Yaskawa INFORM job: X2_38-47,64(2)(90,0).JBI

/JOB
//NAME X2_38-47,64(2)(90,0)
//POS
///NPOS 475,475,475,26,0,0
///TOOL 0
///POSTYPE PULSE
///PULSE
C00000=10776,-116726,-133110,-1428,79202,-268
C00001=117551,-99167,-129064,-14869,107235,-27560
C00002=118060,-97833,-124544,-14759,105287,-27149
C00003=118255,-97731,-122391,-14687,104086,-26936
C00004=118255,-99005,-121658,-14606,103015,-26804
C00005=118252,-98719,-121832,-14623,103261,-26835
C00006=118753,-92238,-119382,-14829,105109,-26899
C00007=118252,-98719,-121832,-14623,103261,-26835
C00008=117548,-101379,-128390,-14732,105732,-27372
C00009=119930,-99721,-129265,-15188,107465,-26816
C00010=120369,-98285,-124713,-15062,105542,-26424
C00011=120537,-98252,-122491,-14975,104264,-26206
C00012=120537,-99415,-121812,-14899,103281,-26083
C00013=120552,-99088,-121997,-14922,103557,-26112
C00014=120983,-92542,-119530,-15124,105413,-26206
C00015=120552,-99088,-121997,-14922,103557,-26112
C00016=119945,-101871,-128593,-15052,105999,-26622
C00017=126449,-117484,-130445,-19479,74849,-30062
C00018=126433,-122162,-123583,-20167,68593,-29001
C00019=126700,-111661,-117040,-20113,69946,-29141
C00020=126798,-108107,-114012,-20160,69935,-29102
C00021=126799,-108400,-113008,-20254,69212,-28975
C00022=126718,-108336,-113627,-20168,69582,-29070
C00023=124486,-105728,-112699,-19107,69790,-29924
C00024=126718,-108336,-113627,-20168,69582,-29070
C00025=121607,-132044,-121280,-18982,61321,-29585
C00026=106120,-105771,-112642,-10491,66484,-36125
C00027=107709,-101450,-111061,-11179,67916,-35692
C00028=106120,-105771,-112642,-10491,66484,-36125
C00029=113778,-131562,-126460,-14735,63009,-32904
C00030=125989,-135705,-128836,-15868,81833,19678
C00031=122637,-125595,-122855,-15098,82666,18409
C00032=121382,-121958,-120533,-14807,82865,17952
C00033=121382,-122071,-118910,-14836,81841,18076
C00034=121382,-121958,-120533,-14807,82865,17952
C00035=106979,-143901,-125029,-2861,68009,11090
C00036=108002,-136905,-123073,-3147,70435,11396
C00037=106979,-143901,-125029,-2861,68009,11090
C00038=130918,-93362,-108301,-23503,98063,21430
C00039=128613,-93045,-108174,-23197,97523,20724
C00040=130918,-93362,-108301,-23503,98063,21430
C00041=136165,-97259,-113946,-24281,100844,22722
C00042=136175,-89641,-119549,-25205,107565,21267
C00043=114744,-130738,-127344,18726,86415,-24127
C00044=118651,-123075,-122041,18017,86194,-22796
C00045=120132,-120263,-119410,17742,85711,-22351
C00046=120132,-120365,-118339,17753,85031,-22450
C00047=120131,-120316,-118616,17749,85218,-22423
C00048=120610,-114014,-116540,17635,86988,-22001
C00049=120131,-120316,-118616,17749,85218,-22423
C00050=120535,-116966,-117470,17658,86102,-22155
C00051=123144,-118008,-117813,17156,85246,-21372
C00052=120535,-116966,-117470,17658,86102,-22155
C00053=115268,-126863,-124750,18631,86672,-23904
C00054=115290,-123417,-132013,18678,92595,-22992
C00055=123593,-125758,-130163,-6995,115060,67946
C00056=111289,-112434,-124190,-9231,117016,63234
C00057=105837,-112853,-120878,-9823,114178,61462
C00058=105837,-113368,-119803,-9744,113264,61541
C00059=105837,-112984,-120626,-9804,113958,61481
C00060=104314,-115180,-121361,-9954,113110,60999
C00061=105837,-112984,-120626,-9804,113958,61481
C00062=140180,-156270,-135194,-3647,103600,74458
C00063=143876,-158808,-133483,-2421,103143,75779
C00064=143876,-157752,-132173,-2418,102880,75785
C00065=143876,-158999,-133717,-2421,103190,75779
C00066=142833,-166242,-135523,-2599,100548,75469
C00067=143876,-158999,-133717,-2421,103190,75779
C00068=138517,-137739,-134524,-3768,114393,73549
C00069=143641,-117492,-131018,-10110,103710,40081
C00070=127017,-112123,-129453,-9078,98380,24722
C00071=128303,-122732,-125182,-9622,82824,11347
C00072=126354,-112603,-118881,-9097,83916,10616
C00073=125631,-108986,-116438,-8904,84188,10357
C00074=125631,-109537,-114964,-8919,83013,10441
C00075=125631,-108986,-116438,-8904,84188,10357
C00076=110037,-120252,-118594,5441,76700,4050
C00077=111650,-115152,-116920,4919,78183,4659
C00078=110037,-120252,-118594,5441,76700,4050
C00079=125797,-107165,-114352,-8951,83863,10435
C00080=123589,-104463,-113383,-8361,84418,9668
C00081=125797,-107165,-114352,-8951,83863,10435
C00082=128447,-120300,-122969,-9661,82730,11402
C00083=128462,-115265,-129707,-9620,89375,10895
C00084=116938,-126430,-125851,12631,81878,-14685
C00085=119474,-116309,-119688,11957,82879,-13726
C00086=120416,-112800,-116898,11714,82830,-13413
C00087=120416,-113088,-115771,11732,82005,-13491
C00088=121130,-109897,-115487,11517,83341,-13125
C00089=121652,-107697,-114715,11371,83913,-12898
C00090=120385,-110630,-116263,11708,83544,-13356
C00091=116898,-126708,-125088,12658,81285,-14759
C00092=116961,-121523,-133241,12544,88781,-13978
C00093=110477,-156196,-127656,40514,54336,-55405
C00094=116757,-147091,-123275,37008,53079,-52657
C00095=119129,-143495,-121504,35581,52690,-51595
C00096=122199,-143523,-121511,34086,51426,-50520
C00097=119129,-143495,-121504,35581,52690,-51595
C00098=121389,-143526,-121523,34489,51757,-50806
C00099=121378,-138155,-118828,34021,52680,-50458
C00100=121389,-143526,-121523,34489,51757,-50806
C00101=121337,-120057,-120260,30579,61379,-47564
C00102=120272,-114318,-116759,30898,62447,-47698
C00103=120254,-119054,-117181,31500,60580,-48280
C00104=120272,-114318,-116759,30898,62447,-47698
C00105=110477,-159292,-131347,40206,54861,-55162
C00106=115322,-144881,-127675,10917,26238,-44128
C00107=131784,-127965,-127002,-28991,89678,-26741
C00108=120831,-123140,-121731,-27130,85392,-29797
C00109=120549,-120601,-118843,-27089,84879,-29783
C00110=120549,-120670,-117777,-27109,84260,-29640
C00111=120517,-120686,-117908,-27101,84315,-29665
C00112=120983,-114470,-115866,-27142,86197,-29928
C00113=120517,-120686,-117908,-27101,84315,-29665
C00114=121539,-130455,-126219,-27290,84728,-29379
C00115=124954,-138498,-133513,-17845,86459,-29447
C00116=125285,-130359,-127302,-17897,86875,-29392
C00117=125412,-127594,-124071,-17925,86361,-29272
C00118=125412,-127626,-123283,-17931,85883,-29202
C00119=125434,-127650,-123440,-17933,85969,-29207
C00120=125746,-120535,-121214,-17972,88215,-29428
C00121=125434,-127650,-123440,-17933,85969,-29207
C00122=125308,-130497,-125835,-17912,85951,-29248
C00123=124977,-138611,-132036,-17860,85542,-29305
C00124=131669,-108309,-130646,-31875,113573,-61343
C00125=139138,-132176,-121475,-37127,109735,-76690
C00126=136347,-141301,-121131,-36509,104575,-76083
C00127=135137,-144527,-120818,-36387,102556,-75910
C00128=135139,-143303,-118803,-36292,102059,-75739
C00129=135137,-144527,-120818,-36387,102556,-75910
C00130=123222,-117207,-112602,-33876,112841,-80142
C00131=123302,-123100,-114500,-33386,111310,-79603
C00132=123222,-117207,-112602,-33876,112841,-80142
C00133=149473,-167599,-122340,-40123,93659,-70303
C00134=145955,-169881,-122827,-40768,91382,-70949
C00135=149473,-167599,-122340,-40123,93659,-70303
C00136=154660,-158984,-124630,-39692,100555,-70658
C00137=145602,-129354,-130944,-11561,117970,-66438
C00138=141571,-135796,-129141,17923,112920,-58745
C00139=145358,-145317,-128855,18021,107261,-58200
C00140=146973,-148537,-128532,18134,105137,-57926
C00141=146977,-147425,-126561,18072,104525,-58019
C00142=146951,-147398,-126788,18082,104677,-58005
C00143=148016,-155121,-128806,18044,101844,-58047
C00144=146951,-147398,-126788,18082,104677,-58005
C00145=147811,-154474,-129578,18071,102659,-57998
C00146=150760,-151393,-128781,18698,103033,-56852
C00147=147811,-154474,-129578,18071,102659,-57998
C00148=142197,-142429,-130522,17697,110344,-58914
C00149=120703,-123129,-132845,-19094,121060,-67264
C00150=120658,-146832,-128060,-18624,118943,-66884
C00151=120634,-158899,-128202,-17585,113113,-65913
C00152=120623,-163194,-128036,-17271,110903,-65572
C00153=120623,-161024,-125795,-17237,110651,-65534
C00154=120562,-161261,-126266,-17282,110799,-65580
C00155=120543,-169070,-128088,-16945,108025,-65171
C00156=120562,-161261,-126266,-17282,110799,-65580
C00157=120603,-145779,-126506,-18564,118536,-66834
C00158=125859,-133715,-124767,-32608,106843,-81797
C00159=122845,-142953,-124347,-32149,101432,-81430
C00160=121547,-146160,-123992,-32074,99345,-81353
C00161=121546,-144979,-121994,-32008,98813,-81200
C00162=109812,-115623,-115113,-28832,111883,-86233
C00163=109420,-121759,-116943,-28463,109962,-85878
C00164=109812,-115651,-114700,-28773,111647,-86169
C00165=136113,-171916,-125823,-37236,88758,-74782
C00166=132431,-173177,-126093,-37775,86796,-75630
C00167=136113,-171916,-125823,-37236,88758,-74782
C00168=141699,-164023,-128432,-36630,95711,-74814
C00169=125872,-133752,-131219,-33440,110189,-40846
C00170=133109,-126295,-132836,-15576,121717,49477
C00171=134095,-144484,-127159,-11413,120192,39245
C00172=134095,-142728,-123587,-11251,118920,39381
C00173=134516,-141672,-122287,-11087,118973,39546
C00174=115660,-122971,-115777,13203,126220,57861
C00175=119843,-134899,-119108,17117,121012,60624
C00176=134151,-138007,-116391,34269,108686,80617
C00177=134077,-138654,-116284,35996,107959,82962
C00178=134074,-140235,-119255,36225,108790,83252
C00179=128746,-104991,-133081,28169,117444,49732
C00180=123335,-90933,-122081,14660,102496,9308
C00181=120623,-92535,-112214,7385,88125,-11837
C00182=120622,-94347,-109953,7392,85821,-11972
C00183=121302,-95773,-109518,7203,84762,-11811
C00184=119347,-92862,-108151,7759,85586,-12396
C00185=120623,-94650,-108957,7399,85059,-12018
C00186=120185,-98069,-104328,-11445,70456,7211
C00187=120621,-97250,-102226,-16251,67423,11647
C00188=120622,-96877,-104163,-16104,68755,11460
C00189=120643,-108357,-118989,-16415,66098,11840
C00190=67024,-106779,-124945,13769,92672,-20129
C00191=67015,-109280,-122780,13735,90127,-20415
C00192=69066,-117370,-123885,13251,86415,-20142
C00193=67301,-111249,-121966,13646,88610,-20491
C00194=67101,-109000,-122679,13716,90193,-20379
C00195=67110,-106486,-124839,13750,92741,-20094
C00196=120616,-103713,-129855,8435,78518,-79847
C00197=120615,-108904,-127553,8566,74477,-80127
C00198=107378,-109964,-123783,23546,74014,-82804
C00199=108339,-95722,-118664,22752,77610,-81754
C00200=115638,-127299,-133424,11228,69296,-82233
C00201=118661,-125998,-116417,35444,53464,-49551
C00202=129777,-134343,-118121,23301,43263,-42347
C00203=129442,-139718,-117663,25605,40832,-43729
C00204=126693,-153141,-115548,34897,36923,-50246
C00205=120532,-119703,-113292,30294,65799,-57942
C00206=118319,-121507,-115012,31110,66714,-58605
C00207=113281,-124998,-118777,32819,69049,-60013
C00208=113467,-117261,-128448,33027,70743,-59318
C00209=117537,-116112,-134646,12805,84442,-25722
C00210=120610,-126431,-125414,-1040,80197,-3464
C00211=120610,-126707,-122448,-1046,78230,-3447
C00212=121742,-127748,-121376,-1361,77053,-3051
C00213=120609,-128006,-121565,-1050,77021,-3438
C00214=120609,-127028,-121195,-1044,77273,-3439
C00215=120354,-127674,-120759,-4484,75447,5144
C00216=120610,-126340,-121533,-4537,76621,5189
C00217=125895,-134934,-128716,-6057,76967,6982
C00218=120648,-124280,-131590,-4464,45149,4941
C00219=120660,-101129,-132257,-5341,102721,45112
C00220=120607,-133883,-126281,-5735,119700,79532
C00221=120606,-133398,-123219,-5634,118073,79618
C00222=123085,-133870,-122397,-4740,117484,80615
C00223=120607,-133916,-122225,-5583,117200,79662
C00224=120605,-135336,-122663,-5559,116742,79683
C00225=119908,-135501,-121613,-12971,116040,68732
C00226=120606,-132780,-121444,-14001,117514,67337
C00227=120606,-133413,-124386,-14219,118956,67146
C00228=118302,-128282,-130929,-25956,92288,30440
C00229=120609,-125694,-119256,-16594,71477,14811
C00230=120609,-125321,-116628,-16727,70109,15005
C00231=120267,-125105,-115730,-16651,69613,14951
C00232=120609,-125784,-120064,8842,76919,-6014
C00233=120609,-126092,-120067,8848,76762,-6022
C00234=120946,-125981,-118164,18196,76467,-19006
C00235=120609,-125456,-118894,18238,77226,-19012
C00236=120610,-125544,-121647,18141,78796,-18775
C00237=120644,-111765,-129409,18832,94472,-5338
C00238=120647,-108820,-131188,26213,120818,60808
C00239=120603,-141811,-125437,24145,112419,84195
C00240=120603,-140407,-122244,23914,111279,83943
C00241=120885,-139622,-121239,23950,111003,83997
C00242=120603,-141924,-124431,0,115210,75490
C00243=120602,-141703,-124653,2,115461,75491
C00244=121293,-137419,-119128,-26325,110161,66441
C00245=120602,-139074,-119094,-30337,107734,65073
C00246=120603,-140473,-121905,-30531,108612,64825
C00247=123038,-137969,-128708,-31970,112888,64779
C00248=147472,-118060,-121113,-40576,103304,81843
C00249=147472,-118630,-118217,-40218,101703,82475
C00250=147472,-118727,-117017,-40094,101093,82713
C00251=147408,-115266,-125424,-616,120610,87255
C00252=147440,-115512,-125518,-608,120541,87267
C00253=147454,-115617,-125558,-7144,119076,75809
C00254=147463,-115686,-125590,-12209,115534,64774
C00255=147467,-115708,-125608,-15036,110623,54333
C00256=147465,-115687,-125611,-15580,106535,46817
C00257=147461,-115654,-125607,-15271,104034,42312
C00258=147458,-115622,-125603,-14500,101619,37854
C00259=147455,-115603,-125598,-14501,101625,37852
C00260=147455,-114670,-126645,-14574,102714,37720
C00261=147454,-112308,-128585,-14752,105047,37432
C00262=120607,-127649,-132770,5702,79300,-5510
C00263=120610,-123519,-126906,5727,77820,-5577
C00264=120610,-124347,-124400,5769,75861,-5668
C00265=121896,-125923,-123599,5365,74477,-5288
C00266=120260,-126985,-123973,12405,76553,-12588
C00267=120608,-127390,-125694,8862,79219,-9976
C00268=120607,-127434,-125218,-886,76106,-6932
C00269=120607,-127109,-124972,1540,76154,-9484
C00270=116410,-121243,-123100,2858,78131,-10867
C00271=112513,-116509,-121595,4066,79794,-12120
C00272=109281,-113129,-120468,5058,81013,-13145
C00273=120610,-123835,-125318,1528,78049,-9462
C00274=120610,-122990,-127374,1521,79748,-9441
C00275=-2000,-133752,-131219,0,47993,0
C00276=63459,-114373,-79771,-19626,40886,-37257
C00277=120535,72123,63468,-4767,55280,-66520
C00278=120830,77643,74299,-5152,51483,-66214
C00279=120946,80397,79380,-5338,49786,-66073
C00280=120946,82340,83558,-5464,48220,-65985
C00281=120946,80397,79380,-5338,49786,-66073
C00282=120262,74330,73734,-4961,50098,-66387
C00283=120723,78845,79280,-5280,49039,-66130
C00284=120262,74330,73734,-4961,50098,-66387
C00285=120141,71846,69055,-4791,51689,-66517
C00286=119837,66739,58851,-4430,55315,-66806
C00287=133022,42927,30487,-538,57153,-74648
C00288=133254,46148,37978,-681,54200,-74537
C00289=133346,47607,41185,-741,52977,-74490
C00290=133347,48340,43676,-753,51820,-74481
C00291=133346,47607,41185,-741,52977,-74490
C00292=132762,43480,38515,-427,52495,-74733
C00293=133123,46716,41988,-628,52023,-74578
C00294=132762,43480,38515,-427,52495,-74733
C00295=132666,42024,35338,-369,53702,-74778
C00296=132425,38795,27897,-232,56620,-74884
C00297=155117,742,-2384,-2320,66217,-73300
C00298=180906,93001,78797,-1706,80780,-74950
C00299=182918,91178,77459,-1890,80713,-74262
C00300=182918,92061,79857,-1895,79691,-74247
C00301=182918,93168,82666,-1899,78530,-74228
C00302=182918,93037,82343,-1899,78661,-74230
C00303=183042,90194,78719,-1906,79434,-74200
C00304=182918,91730,78973,-1891,80062,-74252
C00305=174748,66441,50706,-1110,84503,-77209
C00306=160848,12597,380,297,58397,-81989
C00307=166181,24822,19162,1318,68440,4797
C00308=165629,32403,32901,1529,63893,4538
C00309=165325,34741,37059,1643,62541,4405
C00310=165325,35383,38873,1654,61756,4395
C00311=165325,34741,37059,1643,62541,4405
C00312=165316,38003,40423,1653,62149,4395
C00313=165325,34741,37059,1643,62541,4405
C00314=158615,42058,44677,13811,65940,-11748
C00315=158695,42833,46513,13869,65215,-11806
C00316=159268,43921,47675,13753,64967,-11620
C00317=158695,42064,44447,13779,66066,-11705
C00318=158695,37647,30177,13233,72407,-10974
C00319=159201,26732,24188,1278,51025,-82719
C00320=159224,30548,32077,1320,48132,-82748
C00321=159868,34226,37454,953,46702,-82474
C00322=159868,34770,38966,962,46052,-82480
C00323=159702,29671,32865,1045,47189,-82543
C00324=159324,28280,32585,1288,46650,-82722
C00325=159393,32989,37300,1258,46169,-82698
C00326=159613,30008,32996,1100,47283,-82582
C00327=159229,22535,21884,1275,50287,-82716
C00328=183717,62399,62329,-13487,47753,-71656
C00329=183547,68974,74327,-14313,43831,-71133
C00330=183480,72253,80019,-14758,42056,-70865
C00331=183483,74717,84855,-15260,40402,-70564
C00332=183480,72253,80019,-14758,42056,-70865
C00333=183942,65201,73380,-14911,42587,-70727
C00334=183665,70044,79187,-15050,41486,-70670
C00335=183942,65201,73380,-14911,42587,-70727
C00336=184013,62287,68228,-14508,44220,-70970
C00337=184190,56247,57052,-13734,47916,-71463
C00338=194866,74493,66336,-18454,53556,-67625
C00339=193573,89765,89535,-19520,47162,-66942
C00340=193573,91648,93222,-19932,45935,-66672
C00341=193573,93286,96299,-20287,44943,-66446
C00342=193573,92255,94376,-20065,45559,-66588
C00343=194136,78940,77511,-19269,49033,-67072
C00344=194228,80437,80064,-19546,48302,-66875
C00345=193714,88383,90097,-19926,46207,-66663
C00346=194171,78002,75688,-19109,49654,-67182
C00347=183631,19122,4613,-11412,60722,-73268
C00348=122649,-90706,-82561,19496,61180,-53724
C00349=122649,-90706,-82561,19496,61180,-53724
C00350=146927,-106152,-71782,9593,42642,-76873
C00351=147684,-69879,-51768,13743,41767,-65179
C00352=150199,4793,-22546,4300,98283,-83429
C00353=150319,1938,-15262,4232,92343,-83591
C00354=150367,1184,-14302,4224,91365,-83608
C00355=150367,1240,-12851,4221,90502,-83638
C00356=150367,1184,-14302,4224,91365,-83608
C00357=150123,10711,-6542,4244,91496,-83686
C00358=150277,8779,-6240,4228,90310,-83676
C00359=150175,6887,-7898,4237,90361,-83709
C00360=149968,8102,-7784,4257,90924,-83760
C00361=150441,9583,-10879,4230,93564,-83509
C00362=131878,-32966,-47472,26236,62495,-86167
C00363=135680,-27941,-40403,24709,59747,-85262
C00364=135680,-27934,-39056,24908,58995,-85442
C00365=135680,-27896,-37768,25103,58290,-85615
C00366=135677,-27936,-39177,24874,59064,-85427
C00367=134264,-34276,-43444,25765,58916,-86062
C00368=134265,-34195,-41853,26012,58067,-86277
C00369=135346,-30088,-39110,25338,58118,-85800
C00370=135733,-34145,-44672,24799,59221,-85365
C00371=145616,-30275,-43889,19038,58025,-81528
C00372=147684,-69879,-51768,13743,41767,-65179
C00373=146927,-106152,-71782,9593,42642,-76873
C00374=150216,-104680,-71296,7403,42753,-75254
C00375=181592,-40940,-51538,-10072,64088,-74364
C00376=161871,19225,13725,-11181,66080,-79002
C00377=161452,20882,19453,-11278,63397,-78896
C00378=164352,10606,16407,-20315,52242,-75889
C00379=162815,10479,16392,-19594,51818,-76493
C00380=160145,20957,19678,-10844,63120,-79369
C00381=160561,19267,13917,-10753,65806,-79466
C00382=160561,19267,13917,-10683,67653,-23343
C00383=154925,6937,8528,5000,60577,-30889
C00384=159657,9316,12490,-1477,58995,-24503
C00385=156738,10623,15910,1856,57584,-27775
C00386=156328,10923,16900,2033,57138,-27949
C00387=155501,5675,10762,2341,58239,-28253
C00388=164062,6293,11536,-10601,60711,-458
C00389=163435,22729,32465,-8745,61137,-855
C00390=168216,43762,52548,-18935,71405,19387
C00391=169763,36380,39766,-18709,75622,19280
C00392=165018,20718,26071,-18440,72235,15535
C00393=160304,21163,32931,-8111,30161,-79764
C00394=160077,26796,41073,-8391,28042,-79637
C00395=159587,29219,48591,-14117,21277,-77933
C00396=162103,29346,48721,-18047,21745,-75808
C00397=162103,29346,48721,-18047,21745,-75808
C00398=160812,19418,34049,-13727,25286,-78018
C00399=165374,24294,37670,-31515,32350,-71401
C00400=161014,23173,34950,10300,28145,-85028
C00401=161267,29296,43834,10809,25831,-85265
C00402=163117,31582,50788,6969,18892,-84323
C00403=165058,31936,51150,3284,18732,-82405
C00404=165058,31936,51150,3284,18732,-82405
C00405=165058,26028,37877,2608,23858,-82083
C00406=156219,-6549,3189,13376,29320,-87906
C00407=193662,52178,54811,-23966,35939,-65070
C00408=193395,59348,65976,-25679,32954,-64157
C00409=193846,66406,75330,-27317,31216,-63316
C00410=195732,71420,81412,-29926,30818,-61781
C00411=190088,34040,27543,-17579,42098,-68896
C00412=195743,56061,59163,-26082,35942,-63785
C00413=183848,81700,74678,1498,72719,-73637
C00414=175309,68305,57984,16674,76256,-76182
C00415=174796,71984,66825,17009,72957,-76836
C00416=176911,74218,69518,16737,72030,-76191
C00417=175436,69064,60684,16741,75010,-76311
C00418=157840,39389,32444,18807,80897,-81798
C00419=152544,-11566,-20773,-4534,70818,-69047
C00420=121453,69600,74634,-8596,44521,-67329
C00421=121610,79178,90779,-9562,39584,-66727
C00422=122256,62901,78801,-13281,29449,-64716
C00423=119976,69596,87112,-11678,27131,-65794
C00424=119487,82929,95001,-8292,38695,-67720
C00425=113080,77640,80749,10055,45502,-72493
C00426=113679,80944,85852,9958,44007,-72378
C00427=115090,79143,84432,3405,41517,-71194
C00428=114991,50178,46533,3890,43654,-71191
C00429=130022,56817,59683,7064,48325,-77006
C00430=130464,62791,70833,7260,44523,-77097
C00431=132030,55766,67561,6192,36406,-76838
C00432=136266,49513,60493,2695,37313,-74483
C00433=134997,54946,61777,4491,45732,-74911
C00434=138242,-4678,-14452,2133,61853,-73053
C00435=140332,-41635,-35386,1385,55778,-72457
C00436=125234,-105855,-90971,8573,57832,-78294
C00437=134723,-30987,-43000,16193,82094,73445
C00438=147286,-18641,-32771,-2207,85620,76456
C00439=145565,-8574,-24761,171,91849,76015
C00440=144872,-8220,-24480,237,91860,75784
C00441=148310,-19029,-33055,-2389,85623,76796
C00442=149415,-19533,-33424,-2584,85625,77164
C00443=149671,-4054,-21067,1311,92603,77409
C00444=148276,-3677,-20761,1434,92631,76943
C00445=148276,-3408,-24949,1441,95347,76974
C00446=162074,-26616,-42506,1763,64705,79693
C00447=162070,-24854,-37261,1799,62384,79656
C00448=162588,-20391,-33053,1539,62074,79844
C00449=161725,-20523,-33128,1979,62071,79525
C00450=159769,-24818,-37192,4027,62449,78761
C00451=159682,-26579,-42435,3993,64769,78811
C00452=159749,-26590,-42466,830,64636,81339
C00453=159773,-24828,-37221,834,62313,81331
C00454=157385,-24447,-34130,6743,58116,80693
C00455=158588,-24538,-34197,6069,58011,81159
C00456=162116,-24842,-37231,-1419,62318,82243
C00457=162183,-26603,-42475,-1425,64641,82238
C00458=125234,-105855,-90971,8573,57832,-78294
C00459=122641,-148463,-123471,10002,56262,-79479
C00460=122641,-148463,-123471,10002,56262,-79479
C00461=171100,-2344,-14517,-1298,46918,-78414
C00462=177009,29876,35461,-7963,33075,-74566
C00463=175070,31868,42315,2631,27249,-76698
C00464=178558,34317,44810,-1908,26956,-74189
C00465=176419,28474,30454,-160,33043,-75584
C00466=173102,47124,36593,11518,57062,-77684
C00467=172903,62994,47851,2783,78849,-77249
C00468=172923,63788,52294,3178,77603,-77352
C00469=170832,85464,80401,8251,77478,-78178
C00470=174864,89706,85780,7992,75954,-76876
C00471=176408,69063,51861,3929,81897,-76013
C00472=176687,67050,51974,2579,79340,-76016
C00473=124677,13030,-21056,9614,100342,-34470
C00474=10907,-117335,-90652,18762,63715,59495
BC00000=165804,522273,1075193
BC00001=398158,179848,1075139
BC00002=398158,179848,1075139
BC00003=398158,179848,1075139
BC00004=398158,179848,1075139
BC00005=398158,179848,1075139
BC00006=398158,179848,1075139
BC00007=398158,179848,1075139
BC00008=398158,179848,1075139
BC00009=355141,187784,1075139
BC00010=355141,187784,1075139
BC00011=355141,187784,1075139
BC00012=355141,187784,1075139
BC00013=355141,187784,1075139
BC00014=355141,187784,1075139
BC00015=355141,187784,1075139
BC00016=355141,187784,1075139
BC00017=253971,280733,1075139
BC00018=253971,280733,1075139
BC00019=253971,280733,1075139
BC00020=253971,280733,1075139
BC00021=253971,280733,1075139
BC00022=253971,280733,1075139
BC00023=253971,280733,1075139
BC00024=253971,280733,1075139
BC00025=253971,280733,1075139
BC00026=253971,280733,1075139
BC00027=253971,280733,1075139
BC00028=253971,280733,1075139
BC00029=253971,280733,1075139
BC00030=147021,241254,1075139
BC00031=147021,241254,1075139
BC00032=147021,241254,1075139
BC00033=147021,241254,1075139
BC00034=147021,241254,1075139
BC00035=147021,241254,1075139
BC00036=147021,241254,1075139
BC00037=147021,241254,1075139
BC00038=147021,241254,1075139
BC00039=147021,241254,1075139
BC00040=147021,241254,1075139
BC00041=147021,241254,1075139
BC00042=147021,241254,1075139
BC00043=175602,243488,1075139
BC00044=175602,243488,1075139
BC00045=175602,243488,1075139
BC00046=175602,243488,1075139
BC00047=175602,243488,1075139
BC00048=175602,243488,1075139
BC00049=175602,243488,1075139
BC00050=175602,243488,1075139
BC00051=175602,243488,1075139
BC00052=175602,243488,1075139
BC00053=175602,243488,1075139
BC00054=175602,243488,1075139
BC00055=144296,215160,1075139
BC00056=144296,215160,1075139
BC00057=144296,215160,1075139
BC00058=144296,215160,1075139
BC00059=144296,215160,1075139
BC00060=144296,215160,1075139
BC00061=144296,215160,1075139
BC00062=144296,215160,1075139
BC00063=144296,215160,1075139
BC00064=144296,215160,1075139
BC00065=144296,215160,1075139
BC00066=144296,215160,1075139
BC00067=144296,215160,1075139
BC00068=144296,215160,1075139
BC00069=159912,261457,1075139
BC00070=164424,314586,1075139
BC00071=171018,327464,1075139
BC00072=171018,327464,1075139
BC00073=171018,327464,1075139
BC00074=171018,327464,1075139
BC00075=171018,327464,1075139
BC00076=171018,327464,1075139
BC00077=171018,327464,1075139
BC00078=171018,327464,1075139
BC00079=171018,327464,1075139
BC00080=171018,327464,1075139
BC00081=171018,327464,1075139
BC00082=171018,327464,1075139
BC00083=171018,327464,1075139
BC00084=164722,348126,1075139
BC00085=164722,348126,1075139
BC00086=164722,348126,1075139
BC00087=164722,348126,1075139
BC00088=164722,348126,1075139
BC00089=164722,348126,1075139
BC00090=164722,348126,1075139
BC00091=164722,348126,1075139
BC00092=164722,348126,1075139
BC00093=143323,255421,1075139
BC00094=143323,255421,1075139
BC00095=143323,255421,1075139
BC00096=143323,255421,1075139
BC00097=143323,255421,1075139
BC00098=143323,255421,1075139
BC00099=143323,255421,1075139
BC00100=143323,255421,1075139
BC00101=143323,255421,1075139
BC00102=143323,255421,1075139
BC00103=143323,255421,1075139
BC00104=143323,255421,1075139
BC00105=143323,255421,1075139
BC00106=95176,326084,1075139
BC00107=33051,239015,1075139
BC00108=33051,239015,1075139
BC00109=33051,239015,1075139
BC00110=33051,239015,1075139
BC00111=33051,239015,1075139
BC00112=33051,239015,1075139
BC00113=33051,239015,1075139
BC00114=33051,239015,1075139
BC00115=1592,244787,1075139
BC00116=1592,244787,1075139
BC00117=1592,244787,1075139
BC00118=1592,244787,1075139
BC00119=1592,244787,1075139
BC00120=1592,244787,1075139
BC00121=1592,244787,1075139
BC00122=1592,244787,1075139
BC00123=1592,244787,1075139
BC00124=16444,332290,1075139
BC00125=28284,383081,1075139
BC00126=28284,383081,1075139
BC00127=28284,383081,1075139
BC00128=28284,383081,1075139
BC00129=28284,383081,1075139
BC00130=28284,383081,1075139
BC00131=28284,383081,1075139
BC00132=28284,383081,1075139
BC00133=28284,383081,1075139
BC00134=28284,383081,1075139
BC00135=28284,383081,1075139
BC00136=28284,383081,1075139
BC00137=49933,363253,1075139
BC00138=70307,361243,1075139
BC00139=70307,361243,1075139
BC00140=70307,361243,1075139
BC00141=70307,361243,1075139
BC00142=70307,361243,1075139
BC00143=70307,361243,1075139
BC00144=70307,361243,1075139
BC00145=70307,361243,1075139
BC00146=70307,361243,1075139
BC00147=70307,361243,1075139
BC00148=70307,361243,1075139
BC00149=113384,373634,1075139
BC00150=113384,343814,1075139
BC00151=113384,343814,1075139
BC00152=113384,343814,1075139
BC00153=113384,343814,1075139
BC00154=113384,343814,1075139
BC00155=113384,343814,1075139
BC00156=113384,343814,1075139
BC00157=113384,343814,1075139
BC00158=126163,380629,1075139
BC00159=126163,380629,1075139
BC00160=126163,380629,1075139
BC00161=126163,380629,1075139
BC00162=126163,380629,1075139
BC00163=126163,380629,1075139
BC00164=126163,380629,1075139
BC00165=126163,380629,1075139
BC00166=126163,380629,1075139
BC00167=126163,380629,1075139
BC00168=126163,380629,1075139
BC00169=126163,380629,1075139
BC00170=153244,197421,1075139
BC00171=154878,181155,1075139
BC00172=159551,183681,1075139
BC00173=161025,184477,1075133
BC00174=188164,185165,1075136
BC00175=159382,201380,1075135
BC00176=196155,204160,1075132
BC00177=201120,202214,1075139
BC00178=203654,196593,1075139
BC00179=184090,265203,1075139
BC00180=164129,334283,1075139
BC00181=154120,368924,1075139
BC00182=151898,363919,1075139
BC00183=151009,361917,1075139
BC00184=151009,361917,1075139
BC00185=197558,335778,1075139
BC00186=159988,349936,1075139
BC00187=151141,355258,1075139
BC00188=148277,361304,1075139
BC00189=148277,361304,1075139
BC00190=312259,195594,1075139
BC00191=311963,190251,1075139
BC00192=311844,188113,1075139
BC00193=362717,179281,1075128
BC00194=362836,181418,1075139
BC00195=363132,186762,1075139
BC00196=102779,255305,1075139
BC00197=101436,253332,1075139
BC00198=100899,252542,1075139
BC00199=100899,252542,1075139
BC00200=101410,246391,1075139
BC00201=141499,261853,1075139
BC00202=141499,261853,1075139
BC00203=141499,261853,1075139
BC00204=141499,261852,1075136
BC00205=141499,261853,1075139
BC00206=141499,261853,1075139
BC00207=141499,261853,1075139
BC00208=141499,274005,1075139
BC00209=68111,269753,1075139
BC00210=16814,266781,1075139
BC00211=16546,261584,1075139
BC00212=16439,259506,1075139
BC00213=16439,259506,1075139
BC00214=71877,249918,1075139
BC00215=67448,250953,1075139
BC00216=67006,253063,1075139
BC00217=65899,258340,1075139
BC00218=65899,288131,1075139
BC00219=98307,337973,1075139
BC00220=125063,358885,1075139
BC00221=125778,364300,1075139
BC00222=126063,366466,1075139
BC00223=130842,366450,1075139
BC00224=170092,366314,1075137
BC00225=159428,366441,1075139
BC00226=156853,364418,1075139
BC00227=154110,359318,1075139
BC00228=114676,288419,1075139
BC00229=142986,258877,1075139
BC00230=146299,253666,1075139
BC00231=147625,251582,1075139
BC00232=194925,245639,1075139
BC00233=156825,252253,1075139
BC00234=172687,249256,1075139
BC00235=174276,250992,1075139
BC00236=178251,255331,1075139
BC00237=164902,278776,1075139
BC00238=91091,340629,1075139
BC00239=59682,360606,1075139
BC00240=57241,365786,1075139
BC00241=56264,367859,1075139
BC00242=29820,362432,1075139
BC00243=76738,362270,1075139
BC00244=34590,371298,1075139
BC00245=25837,371005,1075139
BC00246=21253,366566,1075139
BC00247=34673,355700,1075135
BC00248=267722,172731,1075139
BC00249=272714,174556,1075139
BC00250=274711,175286,1075139
BC00251=328692,136963,1075139
BC00252=294146,156358,1075139
BC00253=279419,165219,1075139
BC00254=269323,178854,1075139
BC00255=265414,195151,1075139
BC00256=267320,208388,1075139
BC00257=271316,217638,1075139
BC00258=275010,224166,1075139
BC00259=277506,226556,1075139
BC00260=275846,227409,1075139
BC00261=272525,229113,1075139
BC00262=271699,297736,1073424
BC00263=294810,273775,1075139
BC00264=293529,268177,1075139
BC00265=293016,265937,1075139
BC00266=307027,261102,1075139
BC00267=302570,257740,1075139
BC00268=285679,262491,1075139
BC00269=319740,246081,1075139
BC00270=320984,245484,1075139
BC00271=320984,245484,1075139
BC00272=320984,245484,1075139
BC00273=325754,245581,1075139
BC00274=326738,249882,1075139
BC00275=126163,523905,1075139
BC00276=216710,557083,641270
BC00277=301352,400556,286994
BC00278=301352,400556,286994
BC00279=301352,400556,286994
BC00280=301352,400556,286994
BC00281=301352,400556,286994
BC00282=301352,400556,286994
BC00283=301352,400556,286994
BC00284=301352,400556,286994
BC00285=301352,400556,286994
BC00286=301352,400556,286994
BC00287=314469,400556,277493
BC00288=314469,400556,277493
BC00289=314469,400556,277493
BC00290=314469,400556,277493
BC00291=314469,400556,277493
BC00292=314469,400556,277493
BC00293=314469,400556,277493
BC00294=314469,400556,277493
BC00295=314469,400556,277493
BC00296=314469,400556,277493
BC00297=331599,400556,395859
BC00298=359853,392268,238433
BC00299=359853,392268,238433
BC00300=359853,392268,238433
BC00301=359853,392268,238433
BC00302=359853,392268,238433
BC00303=359853,392268,238433
BC00304=359853,392268,238433
BC00305=343262,398138,316204
BC00306=345835,406354,335171
BC00307=345835,406354,335171
BC00308=345835,406354,335171
BC00309=344242,406354,335171
BC00310=344242,406354,335171
BC00311=344242,406354,335171
BC00312=344242,406354,335171
BC00313=344242,406354,335171
BC00314=344242,406354,335171
BC00315=344242,406354,335171
BC00316=344242,406354,335171
BC00317=344242,406354,335171
BC00318=344242,406354,335171
BC00319=319771,400556,337896
BC00320=319771,400556,337896
BC00321=319771,400556,337896
BC00322=319771,400556,337896
BC00323=319771,400556,337896
BC00324=319771,400556,337896
BC00325=319771,400556,337896
BC00326=319771,400556,337896
BC00327=319771,400556,337896
BC00328=359948,400556,338029
BC00329=359948,400556,338029
BC00330=358355,400556,338029
BC00331=358355,400556,338029
BC00332=358355,400556,338029
BC00333=358355,400556,338029
BC00334=358355,400556,338029
BC00335=358355,400556,338029
BC00336=358355,400556,338029
BC00337=358355,400556,338029
BC00338=365219,400556,270898
BC00339=365219,400556,270898
BC00340=365219,400556,270898
BC00341=365219,400556,270898
BC00342=365219,400556,270898
BC00343=365219,400556,270898
BC00344=365218,400556,270894
BC00345=365218,400556,270894
BC00346=365218,400556,270894
BC00347=365219,411738,375837
BC00348=329511,449778,412801
BC00349=329511,557326,412801
BC00350=219184,520233,311741
BC00351=202274,450326,276450
BC00352=161102,424985,263657
BC00353=161102,424985,263657
BC00354=161102,424985,263657
BC00355=161102,424985,263657
BC00356=161102,424985,263657
BC00357=161102,424985,263657
BC00358=161102,424985,263657
BC00359=161102,424985,263657
BC00360=161102,424985,263657
BC00361=161102,424985,263657
BC00362=144242,432455,148407
BC00363=144242,432455,148407
BC00364=144242,432455,148407
BC00365=144242,432455,148407
BC00366=144243,432453,148404
BC00367=144243,432453,148404
BC00368=144243,432453,148404
BC00369=144243,432453,148404
BC00370=144243,432453,148404
BC00371=179284,432455,148407
BC00372=202274,450326,276450
BC00373=219184,520233,311741
BC00374=365219,520233,600293
BC00375=365219,400556,421118
BC00376=312291,400556,335654
BC00377=312291,400556,335654
BC00378=312291,400556,335654
BC00379=312291,400556,335654
BC00380=312291,400556,335654
BC00381=312291,400556,335654
BC00382=312291,400556,335654
BC00383=312291,400556,335654
BC00384=312291,400556,335654
BC00385=312291,400556,335654
BC00386=312291,400556,335654
BC00387=312291,400556,335654
BC00388=312291,400556,335654
BC00389=312291,400556,375436
BC00390=311759,400169,372248
BC00391=311759,400169,372248
BC00392=312261,400534,445273
BC00393=315262,415157,353191
BC00394=315262,415157,353191
BC00395=315262,415157,353191
BC00396=315262,415157,353191
BC00397=315262,415157,353191
BC00398=315262,415157,353191
BC00399=315262,415157,353191
BC00400=349728,401236,343133
BC00401=349728,401236,343133
BC00402=349728,401236,343133
BC00403=349728,401236,343133
BC00404=349728,401236,343133
BC00405=349728,401236,343133
BC00406=329311,401236,343133
BC00407=366682,400556,290774
BC00408=366682,400556,290774
BC00409=366681,400557,290771
BC00410=366681,400557,290771
BC00411=353522,400557,312772
BC00412=366682,400556,290774
BC00413=341680,400556,335831
BC00414=329114,400556,286060
BC00415=329114,400556,286060
BC00416=329114,400556,286060
BC00417=329114,400556,286060
BC00418=329114,400556,391747
BC00419=306068,400556,345190
BC00420=296056,400556,352007
BC00421=296056,400556,352007
BC00422=296056,400556,352007
BC00423=296056,400556,352007
BC00424=296056,400556,352007
BC00425=296056,400556,305429
BC00426=296056,400556,299166
BC00427=296056,400556,299166
BC00428=296056,400556,299166
BC00429=322956,400556,356242
BC00430=322956,400556,356242
BC00431=322956,400556,356242
BC00432=322956,400556,356242
BC00433=322956,400556,356242
BC00434=323481,404427,418512
BC00435=346006,570548,634248
BC00436=182874,521648,141172
BC00437=138881,416921,238060
BC00438=138881,416921,238060
BC00439=138881,416921,238060
BC00440=138881,416921,238060
BC00441=138881,416921,238060
BC00442=138881,416921,238060
BC00443=147186,418329,239646
BC00444=147186,418329,239646
BC00445=147186,418329,239646
BC00446=187699,415530,182613
BC00447=187699,415530,182613
BC00448=187699,415530,182613
BC00449=187699,415530,182613
BC00450=187699,415530,182613
BC00451=187699,415530,182613
BC00452=187889,415612,182576
BC00453=187889,415612,182576
BC00454=187889,415612,182576
BC00455=187889,415612,182576
BC00456=187889,415612,182576
BC00457=187889,415612,182576
BC00458=182874,521648,141172
BC00459=322956,521648,357949
BC00460=322956,420180,357949
BC00461=348415,400556,248672
BC00462=348415,400556,302439
BC00463=348415,400556,302439
BC00464=348415,400556,302439
BC00465=348415,400556,302439
BC00466=348415,400556,302439
BC00467=339822,400556,351764
BC00468=339562,400556,281997
BC00469=339562,400556,281997
BC00470=339562,400556,281997
BC00471=339562,400556,281997
BC00472=339562,400556,330065
BC00473=340056,504795,481042
BC00474=165804,522273,534000
EC00000=-798156,-183832
EC00001=-798156,-183832
EC00002=-798156,-183832
EC00003=-798156,-183832
EC00004=-798156,-183832
EC00005=-798156,-183832
EC00006=-798156,-183832
EC00007=-798156,-183832
EC00008=-798156,-183832
EC00009=-798156,-183832
EC00010=-798156,-183832
EC00011=-798156,-183832
EC00012=-798156,-183832
EC00013=-798156,-183832
EC00014=-798156,-183832
EC00015=-798156,-183832
EC00016=-798156,-183832
EC00017=-798156,-183832
EC00018=-798156,-183832
EC00019=-798156,-183832
EC00020=-798156,-183832
EC00021=-798156,-183832
EC00022=-798156,-183832
EC00023=-798156,-183832
EC00024=-798156,-183832
EC00025=-798156,-183832
EC00026=-798156,-183832
EC00027=-798156,-183832
EC00028=-798156,-183832
EC00029=-798156,-183832
EC00030=-798156,-183832
EC00031=-798156,-183832
EC00032=-798156,-183832
EC00033=-798156,-183832
EC00034=-798156,-183832
EC00035=-798156,-183832
EC00036=-798156,-183832
EC00037=-798156,-183832
EC00038=-798156,-183832
EC00039=-798156,-183832
EC00040=-798156,-183832
EC00041=-798156,-183832
EC00042=-798156,-183832
EC00043=-798156,-183832
EC00044=-798156,-183832
EC00045=-798156,-183832
EC00046=-798156,-183832
EC00047=-798156,-183832
EC00048=-798156,-183832
EC00049=-798156,-183832
EC00050=-798156,-183832
EC00051=-798156,-183832
EC00052=-798156,-183832
EC00053=-798156,-183832
EC00054=-798156,-183832
EC00055=-798156,-183832
EC00056=-798156,-183832
EC00057=-798156,-183832
EC00058=-798156,-183832
EC00059=-798156,-183832
EC00060=-798156,-183832
EC00061=-798156,-183832
EC00062=-798156,-183832
EC00063=-798156,-183832
EC00064=-798156,-183832
EC00065=-798156,-183832
EC00066=-798156,-183832
EC00067=-798156,-183832
EC00068=-798156,-183832
EC00069=-798156,-183832
EC00070=-798156,-183832
EC00071=-798156,-183832
EC00072=-798156,-183832
EC00073=-798156,-183832
EC00074=-798156,-183832
EC00075=-798156,-183832
EC00076=-798156,-183832
EC00077=-798156,-183832
EC00078=-798156,-183832
EC00079=-798156,-183832
EC00080=-798156,-183832
EC00081=-798156,-183832
EC00082=-798156,-183832
EC00083=-798156,-183832
EC00084=-798156,-183832
EC00085=-798156,-183832
EC00086=-798156,-183832
EC00087=-798156,-183832
EC00088=-798156,-183832
EC00089=-798156,-183832
EC00090=-798156,-183832
EC00091=-798156,-183832
EC00092=-798156,-183832
EC00093=-798156,-183832
EC00094=-798156,-183832
EC00095=-798156,-183832
EC00096=-798156,-183832
EC00097=-798156,-183832
EC00098=-798156,-183832
EC00099=-798156,-183832
EC00100=-798156,-183832
EC00101=-798156,-183832
EC00102=-798156,-183832
EC00103=-798156,-183832
EC00104=-798156,-183832
EC00105=-798156,-183832
EC00106=-798156,-183832
EC00107=-798156,-183832
EC00108=-798156,-183832
EC00109=-798156,-183832
EC00110=-798156,-183832
EC00111=-798156,-183832
EC00112=-798156,-183832
EC00113=-798156,-183832
EC00114=-798156,-183832
EC00115=-798156,-183832
EC00116=-798156,-183832
EC00117=-798156,-183832
EC00118=-798156,-183832
EC00119=-798156,-183832
EC00120=-798156,-183832
EC00121=-798156,-183832
EC00122=-798156,-183832
EC00123=-798156,-183832
EC00124=-798156,-183832
EC00125=-798156,-183832
EC00126=-798156,-183832
EC00127=-798156,-183832
EC00128=-798156,-183832
EC00129=-798156,-183832
EC00130=-798156,-183832
EC00131=-798156,-183832
EC00132=-798156,-183832
EC00133=-798156,-183832
EC00134=-798156,-183832
EC00135=-798156,-183832
EC00136=-798156,-183832
EC00137=-798156,-183832
EC00138=-798156,-183832
EC00139=-798156,-183832
EC00140=-798156,-183832
EC00141=-798156,-183832
EC00142=-798156,-183832
EC00143=-798156,-183832
EC00144=-798156,-183832
EC00145=-798156,-183832
EC00146=-798156,-183832
EC00147=-798156,-183832
EC00148=-798156,-183832
EC00149=-798156,-183832
EC00150=-798156,-183832
EC00151=-798156,-183832
EC00152=-798156,-183832
EC00153=-798156,-183832
EC00154=-798156,-183832
EC00155=-798156,-183832
EC00156=-798156,-183832
EC00157=-798156,-183832
EC00158=-798156,-183832
EC00159=-798156,-183832
EC00160=-798156,-183832
EC00161=-798156,-183832
EC00162=-798156,-183832
EC00163=-798156,-183832
EC00164=-798156,-183832
EC00165=-798156,-183832
EC00166=-798156,-183832
EC00167=-798156,-183832
EC00168=-798156,-183832
EC00169=-798156,-183832
EC00170=-798156,-183832
EC00171=-798156,-183832
EC00172=-798156,-183832
EC00173=-798153,-183835
EC00174=-798155,-183833
EC00175=-798155,-183832
EC00176=-798155,-183833
EC00177=-798156,-183832
EC00178=-798156,-183832
EC00179=-798156,-183832
EC00180=-798156,-183832
EC00181=-798156,-183832
EC00182=-798156,-183832
EC00183=-798156,-183832
EC00184=-798156,-183832
EC00185=-798156,-183832
EC00186=-798156,-183832
EC00187=-798156,-183832
EC00188=-798156,-183832
EC00189=-798156,-183832
EC00190=-798156,-183832
EC00191=-798156,-183832
EC00192=-798156,-183832
EC00193=-798153,-183835
EC00194=-798156,-183832
EC00195=-798156,-183832
EC00196=-798156,-183832
EC00197=-798156,-183832
EC00198=-798156,-183832
EC00199=-798156,-183832
EC00200=-798156,-183832
EC00201=-798156,-183832
EC00202=-798156,-183832
EC00203=-798156,-183832
EC00204=-798155,-183832
EC00205=-798156,-183832
EC00206=-798156,-183832
EC00207=-798156,-183832
EC00208=-798156,-183832
EC00209=-798156,-183832
EC00210=-798156,-183832
EC00211=-798156,-183832
EC00212=-798156,-183832
EC00213=-798156,-183832
EC00214=-798156,-183832
EC00215=-798156,-183832
EC00216=-798156,-183832
EC00217=-798156,-183832
EC00218=-798156,-183832
EC00219=-798156,-183832
EC00220=-798156,-183832
EC00221=-798156,-183832
EC00222=-798156,-183832
EC00223=-798156,-183832
EC00224=-798155,-183832
EC00225=-798156,-183832
EC00226=-798156,-183832
EC00227=-798156,-183832
EC00228=-798156,-183832
EC00229=-798156,-183832
EC00230=-798156,-183832
EC00231=-798156,-183832
EC00232=-798156,-183832
EC00233=-798156,-183832
EC00234=-798156,-183832
EC00235=-798156,-183832
EC00236=-798156,-183832
EC00237=-798156,-183832
EC00238=-798156,-183832
EC00239=-798156,-183832
EC00240=-798156,-183832
EC00241=-798156,-183832
EC00242=-798156,-183832
EC00243=-798156,-183832
EC00244=-798156,-183832
EC00245=-798156,-183832
EC00246=-798156,-183832
EC00247=-798155,-183832
EC00248=-798156,-183832
EC00249=-798156,-183832
EC00250=-798156,-183832
EC00251=-798156,-183832
EC00252=-798156,-183832
EC00253=-798156,-183832
EC00254=-798156,-183832
EC00255=-798156,-183832
EC00256=-798156,-183832
EC00257=-798156,-183832
EC00258=-798156,-183832
EC00259=-798156,-183832
EC00260=-798156,-183832
EC00261=-798156,-183832
EC00262=-798156,-183832
EC00263=-798156,-183832
EC00264=-798156,-183832
EC00265=-798156,-183832
EC00266=-798156,-183832
EC00267=-798156,-183832
EC00268=-798156,-183832
EC00269=-798156,-183832
EC00270=-798156,-183832
EC00271=-798156,-183832
EC00272=-798156,-183832
EC00273=-798156,-183832
EC00274=-798156,-183832
EC00275=-798156,-183832
EC00276=-798156,-183832
EC00277=-798156,-183832
EC00278=-798156,-183832
EC00279=-798156,-183832
EC00280=-798156,-183832
EC00281=-798156,-183832
EC00282=-798156,-183832
EC00283=-798156,-183832
EC00284=-798156,-183832
EC00285=-798156,-183832
EC00286=-798156,-183832
EC00287=-798156,-183832
EC00288=-798156,-183832
EC00289=-798156,-183832
EC00290=-798156,-183832
EC00291=-798156,-183832
EC00292=-798156,-183832
EC00293=-798156,-183832
EC00294=-798156,-183832
EC00295=-798156,-183832
EC00296=-798156,-183832
EC00297=-798156,-183832
EC00298=-798156,-183832
EC00299=-798156,-183832
EC00300=-798156,-183832
EC00301=-798156,-183832
EC00302=-798156,-183832
EC00303=-798156,-183832
EC00304=-798156,-183832
EC00305=-798156,-183832
EC00306=-798156,-183832
EC00307=-798156,-183832
EC00308=-798156,-183832
EC00309=-798156,-183832
EC00310=-798156,-183832
EC00311=-798156,-183832
EC00312=-798156,-183832
EC00313=-798156,-183832
EC00314=-798156,-183832
EC00315=-798156,-183832
EC00316=-798156,-183832
EC00317=-798156,-183832
EC00318=-798156,-183832
EC00319=-798156,-183832
EC00320=-798156,-183832
EC00321=-798156,-183832
EC00322=-798156,-183832
EC00323=-798156,-183832
EC00324=-798156,-183832
EC00325=-798156,-183832
EC00326=-798156,-183832
EC00327=-798156,-183832
EC00328=-798156,-183832
EC00329=-798156,-183832
EC00330=-798156,-183832
EC00331=-798156,-183832
EC00332=-798156,-183832
EC00333=-798156,-183832
EC00334=-798156,-183832
EC00335=-798156,-183832
EC00336=-798156,-183832
EC00337=-798156,-183832
EC00338=-798156,-183832
EC00339=-798156,-183832
EC00340=-798156,-183832
EC00341=-798156,-183832
EC00342=-798156,-183832
EC00343=-798156,-183832
EC00344=-798155,-183832
EC00345=-798155,-183832
EC00346=-798155,-183832
EC00347=-798156,-183832
EC00348=-798156,-183832
EC00349=-798156,-183832
EC00350=-798156,-183832
EC00351=-798156,-183832
EC00352=-798156,-183832
EC00353=-798156,-183832
EC00354=-798156,-183832
EC00355=-798156,-183832
EC00356=-798156,-183832
EC00357=-798156,-183832
EC00358=-798156,-183832
EC00359=-798156,-183832
EC00360=-798156,-183832
EC00361=-798156,-183832
EC00362=-798156,-183832
EC00363=-798156,-183832
EC00364=-798156,-183832
EC00365=-798156,-183832
EC00366=-798155,-183832
EC00367=-798155,-183832
EC00368=-798155,-183832
EC00369=-798155,-183832
EC00370=-798155,-183832
EC00371=-798156,-183832
EC00372=-798156,-183832
EC00373=-798156,-183832
EC00374=-798156,-183832
EC00375=-798156,-183832
EC00376=-798156,-183832
EC00377=-798156,-183832
EC00378=-798156,-183832
EC00379=-798156,-183832
EC00380=-798156,-183832
EC00381=-798156,-183832
EC00382=-798156,-183832
EC00383=-798156,-183832
EC00384=-798156,-183832
EC00385=-798156,-183832
EC00386=-798156,-183832
EC00387=-798156,-183832
EC00388=-798156,-183832
EC00389=-798156,-183832
EC00390=-798156,-183832
EC00391=-798156,-183832
EC00392=-798156,-183832
EC00393=-798156,-183832
EC00394=-798156,-183832
EC00395=-798156,-183832
EC00396=-798156,-183832
EC00397=-798156,-183832
EC00398=-798156,-183832
EC00399=-798156,-183832
EC00400=-798156,-183832
EC00401=-798156,-183832
EC00402=-798156,-183832
EC00403=-798156,-183832
EC00404=-798156,-183832
EC00405=-798156,-183832
EC00406=-798156,-183832
EC00407=-798156,-183832
EC00408=-798156,-183832
EC00409=-798155,-183832
EC00410=-798155,-183832
EC00411=-798155,-183832
EC00412=-798156,-183832
EC00413=-798156,-183832
EC00414=-798156,-183832
EC00415=-798156,-183832
EC00416=-798156,-183832
EC00417=-798156,-183832
EC00418=-798156,-183832
EC00419=-798156,-183832
EC00420=-798156,-183832
EC00421=-798156,-183832
EC00422=-798156,-183832
EC00423=-798156,-183832
EC00424=-798156,-183832
EC00425=-798156,-183832
EC00426=-798156,-183832
EC00427=-798156,-183832
EC00428=-798156,-183832
EC00429=-798156,-183832
EC00430=-798156,-183832
EC00431=-798156,-183832
EC00432=-798156,-183832
EC00433=-798156,-183832
EC00434=-798156,-183832
EC00435=-798156,-183832
EC00436=-798156,-183832
EC00437=-798156,-183832
EC00438=-798156,-183832
EC00439=-798156,-183832
EC00440=-798156,-183832
EC00441=-798156,-183832
EC00442=-798156,-183832
EC00443=-798156,-183832
EC00444=-798156,-183832
EC00445=-798156,-183832
EC00446=-798156,-183832
EC00447=-798156,-183832
EC00448=-798156,-183832
EC00449=-798156,-183832
EC00450=-798156,-183832
EC00451=-798156,-183832
EC00452=-798156,-183832
EC00453=-798156,-183832
EC00454=-798156,-183832
EC00455=-798156,-183832
EC00456=-798156,-183832
EC00457=-798156,-183832
EC00458=-798156,-183832
EC00459=-798156,-183832
EC00460=-798156,-183832
EC00461=-798156,-183832
EC00462=-798156,-183832
EC00463=-798156,-183832
EC00464=-798156,-183832
EC00465=-798156,-183832
EC00466=-798156,-183832
EC00467=-798156,-183832
EC00468=-798156,-183832
EC00469=-798156,-183832
EC00470=-798156,-183832
EC00471=-798156,-183832
EC00472=-798156,-183832
EC00473=-798156,-183832
EC00474=-798156,-183832
///POSTYPE BASE
///RECTAN
///RCONF 0,0,0,0,1,0,0,0,0,0,0,0,0,0,0,0,0,0,0,0,0,0,0,0
P00006=2.006,1.622,-0.565,0.0000,0.0000,0.0000
P00021=0.073,2.058,-0.109,0.0000,0.0000,0.0000
P00022=2.006,1.622,-0.565,0.0000,0.0000,0.0000
///RCONF 0,0,0,0,0,0,0,0,0,0,0,0,0,0,0,0,0,0,0,0,0,0,0,0
P00023=-2.957,-4.083,2.762,0.0000,0.0000,0.0000
P00024=-1.466,-0.226,-0.419,0.0000,0.0000,0.0000
P00025=3.643,0.007,-2.585,0.0000,0.0000,0.0000
P00026=2.644,0.055,-2.583,0.0000,0.0000,0.0000
P00027=2.278,0.099,-4.210,0.0000,0.0000,0.0000
P00028=-1.778,-0.182,-2.050,0.0000,0.0000,0.0000
P00029=1.749,4.006,-0.261,0.0000,0.0000,0.0000
P00030=-0.014,-0.768,0.131,0.0000,0.0000,0.0000
P00031=-0.170,0.039,-0.647,0.0000,0.0000,0.0000
P00032=-0.423,0.157,3.222,0.0000,0.0000,0.0000
P00033=0.854,-1.099,3.047,0.0000,0.0000,0.0000
///RCONF 0,0,0,0,1,0,0,0,0,0,0,0,0,0,0,0,0,0,0,0,0,0,0,0
P00034=-8.151,9.743,-4.393,0.0000,0.0000,0.0000
///RCONF 0,0,0,0,0,0,0,0,0,0,0,0,0,0,0,0,0,0,0,0,0,0,0,0
P00042=-0.220,0.371,-0.613,0.0000,0.0000,0.0000
P00043=-0.179,-5.890,-3.227,0.0000,0.0000,0.0000
P00044=-8.560,-7.557,-5.232,0.0000,0.0000,0.0000
P00045=-8.836,-6.632,-1.438,0.0000,0.0000,0.0000
P00046=-7.725,-0.107,-2.878,0.0000,0.0000,0.0000
///RCONF 0,1,0,0,0,0,0,0,0,0,0,0,0,0,0,0,0,0,0,0,0,0,0,0
P00047=0.052,4.745,-6.175,0.0000,0.0000,0.0000
///RCONF 0,0,0,0,0,0,0,0,0,0,0,0,0,0,0,0,0,0,0,0,0,0,0,0
P00048=-10.315,0.035,-3.101,0.0000,0.0000,0.0000
P00049=-9.638,1.690,-2.627,0.0000,0.0000,0.0000
P00051=-5.945,4.696,-10.293,0.0000,0.0000,0.0000
P00060=1524.284,698.404,-261.973,-0.4635,36.8346,-1.2388
P00091=1.048,0.648,3.624,0.0000,0.0000,0.0000
//INST
///DATE 2024/12/18 17:03
///ATTR SC,RW
///GROUP1 RB1,BS1
///GROUP2 ST1
NOP
'X2_38-47,64(2)(90,0)
'Down
MOVJ C00000 BC00000 VJ=100.00  +MOVJ EC00000 VJ=100.00
'Up
'Path S4602
SFTOF3D
MOVJ C00001 BC00001 VJ=100.00  +MOVJ EC00001 VJ=100.00
MOVL C00002 BC00002 V=800.0  +MOVJ EC00002 VJ=100.00
SMOVL C00003 BC00003 V=166.7  +MOVJ EC00003
SREFP 3 C00004 BC00004  +REFP EC00004
CALL JOB:SEARCH-R1-S13D
SET P021 P006
SFTON3D P021
SMOVL C00005 BC00005 V=166.7  +MOVJ EC00005
SREFP 3 C00006 BC00006  +REFP EC00006
CALL JOB:SEARCH-R1-S13D
SET P021 P006
SFTON3D P021
SMOVL C00007 BC00007 V=166.7  +MOVJ EC00007
MOVL C00008 BC00008 V=1000.0  +MOVJ EC00008 VJ=100.00
'EndPath S4602
'Path S4603
SFTOF3D
MOVJ C00009 BC00009 VJ=100.00  +MOVJ EC00009 VJ=100.00
MOVL C00010 BC00010 V=800.0  +MOVJ EC00010 VJ=100.00
SMOVL C00011 BC00011 V=166.7  +MOVJ EC00011
SREFP 3 C00012 BC00012  +REFP EC00012
CALL JOB:SEARCH-R1-S13D
SET P022 P006
SFTON3D P022
SMOVL C00013 BC00013 V=166.7  +MOVJ EC00013
SREFP 3 C00014 BC00014  +REFP EC00014
CALL JOB:SEARCH-R1-S13D
SET P022 P006
SFTON3D P022
SMOVL C00015 BC00015 V=166.7  +MOVJ EC00015
MOVL C00016 BC00016 V=1000.0  +MOVJ EC00016 VJ=100.00
'EndPath S4603
'Path S4604
SFTOF3D
MOVJ C00017 BC00017 VJ=100.00  +MOVJ EC00017 VJ=100.00
MOVJ C00018 BC00018 VJ=100.00  +MOVJ EC00018 VJ=100.00
MOVL C00019 BC00019 V=800.0  +MOVJ EC00019 VJ=100.00
SMOVL C00020 BC00020 V=166.7  +MOVJ EC00020
SREFP 3 C00021 BC00021  +REFP EC00021
CALL JOB:SEARCH-R1-S13D
SET P023 P006
SFTON3D P023
SMOVL C00022 BC00022 V=166.7  +MOVJ EC00022
SREFP 3 C00023 BC00023  +REFP EC00023
CALL JOB:SEARCH-R1-S13D
SET P023 P006
SFTON3D P023
SMOVL C00024 BC00024 V=166.7  +MOVJ EC00024
SMOVL C00025 BC00025 V=333.3  +MOVJ EC00025
SMOVL C00026 BC00026 V=333.3  +MOVJ EC00026
SREFP 3 C00027 BC00027  +REFP EC00027
CALL JOB:SEARCH-R1-S13D
SET P023 P006
SFTON3D P023
SMOVL C00028 BC00028 V=166.7  +MOVJ EC00028
MOVL C00029 BC00029 V=1000.0  +MOVJ EC00029 VJ=100.00
'EndPath S4604
'Path S4605
SFTOF3D
MOVJ C00030 BC00030 VJ=100.00  +MOVJ EC00030 VJ=100.00
MOVL C00031 BC00031 V=800.0  +MOVJ EC00031 VJ=100.00
SMOVL C00032 BC00032 V=166.7  +MOVJ EC00032
SREFP 3 C00033 BC00033  +REFP EC00033
CALL JOB:SEARCH-R1-S13D
SET P024 P006
SFTON3D P024
SMOVL C00034 BC00034 V=166.7  +MOVJ EC00034
SMOVL C00035 BC00035 V=166.7  +MOVJ EC00035
SREFP 3 C00036 BC00036  +REFP EC00036
CALL JOB:SEARCH-R1-S13D
SET P024 P006
SFTON3D P024
SMOVL C00037 BC00037 V=166.7  +MOVJ EC00037
SMOVL C00038 BC00038 V=166.7  +MOVJ EC00038
SREFP 3 C00039 BC00039  +REFP EC00039
CALL JOB:SEARCH-R1-S13D
SET P024 P006
SFTON3D P024
SMOVL C00040 BC00040 V=166.7  +MOVJ EC00040
MOVL C00041 BC00041 V=1000.0  +MOVJ EC00041 VJ=100.00
MOVL C00042 BC00042 V=1000.0  +MOVJ EC00042 VJ=100.00
'EndPath S4605
'Path S4606
SFTOF3D
MOVJ C00043 BC00043 VJ=100.00  +MOVJ EC00043 VJ=100.00
MOVL C00044 BC00044 V=800.0  +MOVJ EC00044 VJ=100.00
SMOVL C00045 BC00045 V=166.7  +MOVJ EC00045
SREFP 3 C00046 BC00046  +REFP EC00046
CALL JOB:SEARCH-R1-S13D
SET P025 P006
SFTON3D P025
SMOVL C00047 BC00047 V=166.7  +MOVJ EC00047
SREFP 3 C00048 BC00048  +REFP EC00048
CALL JOB:SEARCH-R1-S13D
SET P025 P006
SFTON3D P025
SMOVL C00049 BC00049 V=166.7  +MOVJ EC00049
SMOVL C00050 BC00050 V=166.7  +MOVJ EC00050
SREFP 3 C00051 BC00051  +REFP EC00051
CALL JOB:SEARCH-R1-S13D
SET P025 P006
SFTON3D P025
SMOVL C00052 BC00052 V=166.7  +MOVJ EC00052
MOVL C00053 BC00053 V=1000.0  +MOVJ EC00053 VJ=100.00
MOVL C00054 BC00054 V=1000.0  +MOVJ EC00054 VJ=100.00
'EndPath S4606
'Path S4607
SFTOF3D
MOVJ C00055 BC00055 VJ=100.00  +MOVJ EC00055 VJ=100.00
MOVL C00056 BC00056 V=800.0  +MOVJ EC00056 VJ=100.00
SMOVL C00057 BC00057 V=166.7  +MOVJ EC00057
SREFP 3 C00058 BC00058  +REFP EC00058
CALL JOB:SEARCH-R1-S13D
SET P026 P006
SFTON3D P026
SMOVL C00059 BC00059 V=166.7  +MOVJ EC00059
SREFP 3 C00060 BC00060  +REFP EC00060
CALL JOB:SEARCH-R1-S13D
SET P026 P006
SFTON3D P026
SMOVL C00061 BC00061 V=166.7  +MOVJ EC00061
MOVL C00062 BC00062 V=1000.0  +MOVJ EC00062 VJ=100.00
SFTOF3D
SMOVL C00063 BC00063 V=166.7  +MOVJ EC00063
SREFP 3 C00064 BC00064  +REFP EC00064
CALL JOB:SEARCH-R1-S13D
SET P091 P006
SFTON3D P091
SMOVL C00065 BC00065 V=166.7  +MOVJ EC00065
SREFP 3 C00066 BC00066  +REFP EC00066
CALL JOB:SEARCH-R1-S13D
SET P091 P006
SFTON3D P091
SMOVL C00067 BC00067 V=166.7  +MOVJ EC00067
SMOVL C00068 BC00068 V=500.0  +MOVJ EC00068
'EndPath S4607
MOVJ C00069 BC00069 VJ=100.00  +MOVJ EC00069 VJ=100.00
MOVJ C00070 BC00070 VJ=100.00  +MOVJ EC00070 VJ=100.00
'Path S4608
SFTOF3D
MOVJ C00071 BC00071 VJ=100.00  +MOVJ EC00071 VJ=100.00
MOVL C00072 BC00072 V=800.0  +MOVJ EC00072 VJ=100.00
SMOVL C00073 BC00073 V=166.7  +MOVJ EC00073
SREFP 3 C00074 BC00074  +REFP EC00074
CALL JOB:SEARCH-R1-S13D
SET P027 P006
SFTON3D P027
SMOVL C00075 BC00075 V=166.7  +MOVJ EC00075
SMOVL C00076 BC00076 V=166.7  +MOVJ EC00076
SREFP 3 C00077 BC00077  +REFP EC00077
CALL JOB:SEARCH-R1-S13D
SET P027 P006
SFTON3D P027
SMOVL C00078 BC00078 V=166.7  +MOVJ EC00078
SMOVL C00079 BC00079 V=166.7  +MOVJ EC00079
SREFP 3 C00080 BC00080  +REFP EC00080
CALL JOB:SEARCH-R1-S13D
SET P027 P006
SFTON3D P027
SMOVL C00081 BC00081 V=166.7  +MOVJ EC00081
MOVL C00082 BC00082 V=1000.0  +MOVJ EC00082 VJ=100.00
MOVL C00083 BC00083 V=1000.0  +MOVJ EC00083 VJ=100.00
'EndPath S4608
'Path S4609
SFTOF3D
MOVJ C00084 BC00084 VJ=100.00  +MOVJ EC00084 VJ=100.00
MOVL C00085 BC00085 V=800.0  +MOVJ EC00085 VJ=100.00
SMOVL C00086 BC00086 V=166.7  +MOVJ EC00086
SREFP 3 C00087 BC00087  +REFP EC00087
CALL JOB:SEARCH-R1-S13D
SET P028 P006
SFTON3D P028
SMOVL C00088 BC00088 V=166.7  +MOVJ EC00088
SREFP 3 C00089 BC00089  +REFP EC00089
CALL JOB:SEARCH-R1-S13D
SET P028 P006
SFTON3D P028
SMOVL C00090 BC00090 V=250.0  +MOVJ EC00090
MOVL C00091 BC00091 V=1000.0  +MOVJ EC00091 VJ=100.00
'EndPath S4609
MOVJ C00092 BC00092 VJ=100.00  +MOVJ EC00092 VJ=100.00
'Path S4882
SFTOF3D
MOVJ C00093 BC00093 VJ=100.00  +MOVJ EC00093 VJ=100.00
MOVL C00094 BC00094 V=800.0  +MOVJ EC00094 VJ=100.00
SMOVL C00095 BC00095 V=166.7  +MOVJ EC00095
SREFP 3 C00096 BC00096  +REFP EC00096
CALL JOB:SEARCH-R1-S13D
SET P060 P006
SFTON3D P060
SMOVL C00097 BC00097 V=166.7  +MOVJ EC00097
SMOVL C00098 BC00098 V=166.7  +MOVJ EC00098
SREFP 3 C00099 BC00099  +REFP EC00099
CALL JOB:SEARCH-R1-S13D
SET P060 P006
SFTON3D P060
SMOVL C00100 BC00100 V=166.7  +MOVJ EC00100
SMOVL C00101 BC00101 V=333.3  +MOVJ EC00101
SMOVL C00102 BC00102 V=166.7  +MOVJ EC00102
SREFP 3 C00103 BC00103  +REFP EC00103
CALL JOB:SEARCH-R1-S13D
SET P060 P006
SFTON3D P060
SMOVL C00104 BC00104 V=166.7  +MOVJ EC00104
MOVL C00105 BC00105 V=1000.0  +MOVJ EC00105 VJ=100.00
'EndPath S4882
MOVJ C00106 BC00106 VJ=100.00  +MOVJ EC00106 VJ=100.00
'Path S4610
SFTOF3D
MOVJ C00107 BC00107 VJ=100.00  +MOVJ EC00107 VJ=100.00
MOVL C00108 BC00108 V=800.0  +MOVJ EC00108 VJ=100.00
SMOVL C00109 BC00109 V=166.7  +MOVJ EC00109
SREFP 3 C00110 BC00110  +REFP EC00110
CALL JOB:SEARCH-R1-S13D
SET P029 P006
SFTON3D P029
SMOVL C00111 BC00111 V=166.7  +MOVJ EC00111
SREFP 3 C00112 BC00112  +REFP EC00112
CALL JOB:SEARCH-R1-S13D
SET P029 P006
SFTON3D P029
SMOVL C00113 BC00113 V=166.7  +MOVJ EC00113
MOVL C00114 BC00114 V=1000.0  +MOVJ EC00114 VJ=100.00
'EndPath S4610
'Path S4611
SFTOF3D
MOVJ C00115 BC00115 VJ=100.00  +MOVJ EC00115 VJ=100.00
MOVL C00116 BC00116 V=800.0  +MOVJ EC00116 VJ=100.00
SMOVL C00117 BC00117 V=166.7  +MOVJ EC00117
SREFP 3 C00118 BC00118  +REFP EC00118
CALL JOB:SEARCH-R1-S13D
SET P030 P006
SFTON3D P030
SMOVL C00119 BC00119 V=166.7  +MOVJ EC00119
SREFP 3 C00120 BC00120  +REFP EC00120
CALL JOB:SEARCH-R1-S13D
SET P030 P006
SFTON3D P030
SMOVL C00121 BC00121 V=166.7  +MOVJ EC00121
MOVL C00122 BC00122 V=800.0  +MOVJ EC00122 VJ=100.00
MOVL C00123 BC00123 V=1000.0  +MOVJ EC00123 VJ=100.00
'EndPath S4611
MOVJ C00124 BC00124 VJ=100.00  +MOVJ EC00124 VJ=100.00
'Path S4612
SFTOF3D
MOVJ C00125 BC00125 VJ=100.00  +MOVJ EC00125 VJ=100.00
MOVL C00126 BC00126 V=800.0  +MOVJ EC00126 VJ=100.00
SMOVL C00127 BC00127 V=166.7  +MOVJ EC00127
SREFP 3 C00128 BC00128  +REFP EC00128
CALL JOB:SEARCH-R1-S13D
SET P031 P006
SFTON3D P031
SMOVL C00129 BC00129 V=166.7  +MOVJ EC00129
SMOVL C00130 BC00130 V=166.7  +MOVJ EC00130
SREFP 3 C00131 BC00131  +REFP EC00131
CALL JOB:SEARCH-R1-S13D
SET P031 P006
SFTON3D P031
SMOVL C00132 BC00132 V=166.7  +MOVJ EC00132
SMOVL C00133 BC00133 V=166.7  +MOVJ EC00133
SREFP 3 C00134 BC00134  +REFP EC00134
CALL JOB:SEARCH-R1-S13D
SET P031 P006
SFTON3D P031
SMOVL C00135 BC00135 V=166.7  +MOVJ EC00135
MOVL C00136 BC00136 V=1000.0  +MOVJ EC00136 VJ=100.00
'EndPath S4612
MOVJ C00137 BC00137 VJ=100.00  +MOVJ EC00137 VJ=100.00
'Path S4613
SFTOF3D
MOVJ C00138 BC00138 VJ=100.00  +MOVJ EC00138 VJ=100.00
MOVL C00139 BC00139 V=800.0  +MOVJ EC00139 VJ=100.00
SMOVL C00140 BC00140 V=166.7  +MOVJ EC00140
SREFP 3 C00141 BC00141  +REFP EC00141
CALL JOB:SEARCH-R1-S13D
SET P032 P006
SFTON3D P032
SMOVL C00142 BC00142 V=166.7  +MOVJ EC00142
SREFP 3 C00143 BC00143  +REFP EC00143
CALL JOB:SEARCH-R1-S13D
SET P032 P006
SFTON3D P032
SMOVL C00144 BC00144 V=166.7  +MOVJ EC00144
SMOVL C00145 BC00145 V=166.7  +MOVJ EC00145
SREFP 3 C00146 BC00146  +REFP EC00146
CALL JOB:SEARCH-R1-S13D
SET P032 P006
SFTON3D P032
SMOVL C00147 BC00147 V=166.7  +MOVJ EC00147
MOVL C00148 BC00148 V=1000.0  +MOVJ EC00148 VJ=100.00
'EndPath S4613
MOVJ C00149 BC00149 VJ=100.00  +MOVJ EC00149 VJ=100.00
'Path S4614
SFTOF3D
MOVJ C00150 BC00150 VJ=100.00  +MOVJ EC00150 VJ=100.00
MOVL C00151 BC00151 V=800.0  +MOVJ EC00151 VJ=100.00
SMOVL C00152 BC00152 V=166.7  +MOVJ EC00152
SREFP 3 C00153 BC00153  +REFP EC00153
CALL JOB:SEARCH-R1-S13D
SET P033 P006
SFTON3D P033
SMOVL C00154 BC00154 V=166.7  +MOVJ EC00154
SREFP 3 C00155 BC00155  +REFP EC00155
CALL JOB:SEARCH-R1-S13D
SET P033 P006
SFTON3D P033
SMOVL C00156 BC00156 V=166.7  +MOVJ EC00156
MOVL C00157 BC00157 V=1000.0  +MOVJ EC00157 VJ=100.00
'EndPath S4614
'Path S4615
SFTOF3D
MOVJ C00158 BC00158 VJ=100.00  +MOVJ EC00158 VJ=100.00
MOVL C00159 BC00159 V=800.0  +MOVJ EC00159 VJ=100.00
SMOVL C00160 BC00160 V=166.7  +MOVJ EC00160
SREFP 3 C00161 BC00161  +REFP EC00161
CALL JOB:SEARCH-R1-S13D
SET P034 P006
SFTON3D P034
SMOVL C00162 BC00162 V=166.7  +MOVJ EC00162
SREFP 3 C00163 BC00163  +REFP EC00163
CALL JOB:SEARCH-R1-S13D
SET P034 P006
SFTON3D P034
SMOVL C00164 BC00164 V=166.7  +MOVJ EC00164
SMOVL C00165 BC00165 V=166.7  +MOVJ EC00165
SREFP 3 C00166 BC00166  +REFP EC00166
CALL JOB:SEARCH-R1-S13D
SET P034 P006
SFTON3D P034
SMOVL C00167 BC00167 V=166.7  +MOVJ EC00167
MOVL C00168 BC00168 V=1000.0  +MOVJ EC00168 VJ=100.00
'EndPath S4615
MOVJ C00169 BC00169 VJ=100.00  +MOVJ EC00169 VJ=100.00
MOVJ C00170 BC00170 VJ=100.00  +MOVJ EC00170 VJ=100.00
'Path W4616
SFTOF3D
SFTON3D P026
MOVJ C00171 BC00171 VJ=100.00  +MOVJ EC00171 VJ=100.00
SMOVL C00172 BC00172 V=800.0  +MOVJ EC00172
'POPRAWIC!!!!
SMOVL C00173 BC00173 V=166.7 PL=0  +MOVJ EC00173
MACRO1 MJ#(0) ARGF21
ARCON
SWVON WEV#(100)
SMOVL C00174 BC00174 V=9.2  +MOVJ EC00174
SFTON3D P091
SMOVL C00175 BC00175 V=9.2  +MOVJ EC00175
SMOVL C00176 BC00176 V=9.2  +MOVJ EC00176
SWVOF
ARCOF
SMOVL C00177 BC00177 V=800.0  +MOVJ EC00177
SMOVL C00178 BC00178 V=1000.0  +MOVJ EC00178
SFTOF3D
'EndPath W4616
MOVJ C00179 BC00179 VJ=100.00  +MOVJ EC00179 VJ=100.00
'Path W4617
SFTOF3D
SFTON3D P028
MOVJ C00180 BC00180 VJ=100.00  +MOVJ EC00180 VJ=100.00
MOVJ C00181 BC00181 VJ=100.00  +MOVJ EC00181 VJ=100.00
SMOVL C00182 BC00182 V=800.0  +MOVJ EC00182
SMOVL C00183 BC00183 V=150.0 PL=0  +MOVJ EC00183
ARCON
SWVON WEV#(100)
MOVL C00184 BC00184 V=9.2  +MOVJ EC00184 VJ=100.00
SFTON3D P027
SMOVL C00185 BC00185 V=9.2  +MOVJ EC00185
SMOVL C00186 BC00186 V=9.2  +MOVJ EC00186
ARCOF
SWVOF
SMOVL C00187 BC00187 V=800.0  +MOVJ EC00187
SMOVL C00188 BC00188 V=1000.0  +MOVJ EC00188
SFTOF3D
'EndPath W4617
MOVJ C00189 BC00189 VJ=100.00  +MOVJ EC00189 VJ=100.00
'Path W4618
SFTOF3D
SFTON3D P022
MOVJ C00190 BC00190 VJ=100.00  +MOVJ EC00190 VJ=100.00
SMOVL C00191 BC00191 V=800.0  +MOVJ EC00191
SMOVL C00192 BC00192 V=150.0 PL=0  +MOVJ EC00192
MACRO1 MJ#(0) ARGF9
ARCON
SWVON WEV#(60)
SFTON3D P021
SMOVL C00193 BC00193 V=10.0  +MOVJ EC00193
ARCOF
SWVOF
SMOVL C00194 BC00194 V=800.0  +MOVJ EC00194
SMOVL C00195 BC00195 V=1000.0  +MOVJ EC00195
SFTOF3D
'EndPath W4618
'Path W4883
SFTOF3D
SFTON3D P060
MOVJ C00196 BC00196 VJ=100.00  +MOVJ EC00196 VJ=100.00
SMOVL C00197 BC00197 V=800.0  +MOVJ EC00197
SMOVL C00198 BC00198 V=150.0 PL=0  +MOVJ EC00198
ARCON
SMOVL C00199 BC00199 V=10.0  +MOVJ EC00199
ARCOF
SMOVL C00200 BC00200 V=800.0  +MOVJ EC00200
SFTOF3D
'EndPath W4883
'Path W4884
SFTOF3D
SFTON3D P060
SMOVL C00201 BC00201 V=800.0  +MOVJ EC00201
SMOVL C00202 BC00202 V=150.0 PL=0  +MOVJ EC00202
ARCON
SMOVL C00203 BC00203 V=10.0  +MOVJ EC00203
SMOVL C00204 BC00204 V=10.0  +MOVJ EC00204
SMOVL C00205 BC00205 V=10.0  +MOVJ EC00205
ARCOF
SMOVL C00206 BC00206 V=800.0  +MOVJ EC00206
SMOVL C00207 BC00207 V=1000.0  +MOVJ EC00207
SFTOF3D
'EndPath W4884
MOVJ C00208 BC00208 VJ=100.00  +MOVJ EC00208 VJ=100.00
'Path W4619
SFTOF3D
SFTON3D P030
MOVJ C00209 BC00209 VJ=100.00  +MOVJ EC00209 VJ=100.00
MOVJ C00210 BC00210 VJ=100.00  +MOVJ EC00210 VJ=100.00
SMOVL C00211 BC00211 V=800.0  +MOVJ EC00211
SMOVL C00212 BC00212 V=150.0 PL=0  +MOVJ EC00212
ARCON
MOVL C00213 BC00213 V=10.0  +MOVJ EC00213 VJ=100.00
SFTON3D P029
SMOVL C00214 BC00214 V=10.0  +MOVJ EC00214
SMOVL C00215 BC00215 V=10.0  +MOVJ EC00215
ARCOF
SMOVL C00216 BC00216 V=800.0  +MOVJ EC00216
SMOVL C00217 BC00217 V=1000.0  +MOVJ EC00217
SFTOF3D
'EndPath W4619
MOVJ C00218 BC00218 VJ=100.00  +MOVJ EC00218 VJ=100.00
MOVJ C00219 BC00219 VJ=100.00  +MOVJ EC00219 VJ=100.00
'Path W4620
SFTOF3D
SFTON3D P033
MOVJ C00220 BC00220 VJ=100.00  +MOVJ EC00220 VJ=100.00
SMOVL C00221 BC00221 V=800.0  +MOVJ EC00221
SMOVL C00222 BC00222 V=166.7 PL=0  +MOVJ EC00222
ARCON
SMOVL C00223 BC00223 V=9.2  +MOVJ EC00223
SFTON3D P034
SMOVL C00224 BC00224 V=9.2  +MOVJ EC00224
SMOVL C00225 BC00225 V=9.2  +MOVJ EC00225
ARCOF
SMOVL C00226 BC00226 V=800.0  +MOVJ EC00226
SMOVL C00227 BC00227 V=1000.0  +MOVJ EC00227
SFTOF3D
'EndPath W4620
MOVJ C00228 BC00228 VJ=100.00  +MOVJ EC00228 VJ=100.00
'Path W4621
SFTOF3D
SFTON3D P024
MOVJ C00229 BC00229 VJ=100.00  +MOVJ EC00229 VJ=100.00
SMOVL C00230 BC00230 V=800.0  +MOVJ EC00230
SMOVL C00231 BC00231 V=166.7 PL=0  +MOVJ EC00231
ARCON
SMOVL C00232 BC00232 V=10.0  +MOVJ EC00232
SFTON3D P025
SMOVL C00233 BC00233 V=10.0  +MOVJ EC00233
SMOVL C00234 BC00234 V=10.0  +MOVJ EC00234
ARCOF
SMOVL C00235 BC00235 V=800.0  +MOVJ EC00235
SMOVL C00236 BC00236 V=1000.0  +MOVJ EC00236
SFTOF3D
'EndPath W4621
MOVJ C00237 BC00237 VJ=100.00  +MOVJ EC00237 VJ=100.00
MOVJ C00238 BC00238 VJ=100.00  +MOVJ EC00238 VJ=100.00
'Path W4622
SFTOF3D
SFTON3D P032
MOVJ C00239 BC00239 VJ=100.00  +MOVJ EC00239 VJ=100.00
SMOVL C00240 BC00240 V=800.0  +MOVJ EC00240
SMOVL C00241 BC00241 V=166.7 PL=0  +MOVJ EC00241
ARCON
SMOVL C00242 BC00242 V=9.2  +MOVJ EC00242
SFTON3D P031
SMOVL C00243 BC00243 V=9.2  +MOVJ EC00243
SMOVL C00244 BC00244 V=9.2  +MOVJ EC00244
ARCOF
SMOVL C00245 BC00245 V=800.0  +MOVJ EC00245
SMOVL C00246 BC00246 V=1000.0  +MOVJ EC00246
SFTOF3D
'EndPath W4622
'Path W4623
SFTOF3D
SFTON3D P023
MOVJ C00247 BC00247 VJ=100.00  +MOVJ EC00247 VJ=100.00
JUMP *VVP
MOVJ C00248 BC00248 VJ=100.00  +MOVJ EC00248 VJ=100.00
SMOVL C00249 BC00249 V=800.0  +MOVJ EC00249
SMOVL C00250 BC00250 V=166.7 PL=0  +MOVJ EC00250
'ARCON DO SPRAWDZENIA
PAUSE
SMOVL C00251 BC00251 V=10.0  +MOVJ EC00251
SMOVL C00252 BC00252 V=10.0  +MOVJ EC00252
SMOVL C00253 BC00253 V=10.0  +MOVJ EC00253
SMOVL C00254 BC00254 V=10.0  +MOVJ EC00254
SMOVL C00255 BC00255 V=10.0  +MOVJ EC00255
SMOVL C00256 BC00256 V=10.0  +MOVJ EC00256
SMOVL C00257 BC00257 V=10.0  +MOVJ EC00257
SMOVL C00258 BC00258 V=10.0  +MOVJ EC00258
SMOVL C00259 BC00259 V=10.0  +MOVJ EC00259
ARCOF
SMOVL C00260 BC00260 V=800.0  +MOVJ EC00260
SMOVL C00261 BC00261 V=1000.0  +MOVJ EC00261
SFTOF3D
'EndPath W4623
'Path W4624
*VVP
MOVJ C00262 BC00262 VJ=100.00  +MOVJ EC00262 VJ=100.00
SFTOF3D
SFTON3D P023
MOVJ C00263 BC00263 VJ=100.00  +MOVJ EC00263 VJ=100.00
SMOVL C00264 BC00264 V=800.0  +MOVJ EC00264
SMOVL C00265 BC00265 V=150.0 PL=0  +MOVJ EC00265
ARCON
SMOVL C00266 BC00266 V=8.3  +MOVJ EC00266
SMOVL C00267 BC00267 V=8.3  +MOVJ EC00267
SMOVL C00268 BC00268 V=8.3  +MOVJ EC00268
SMOVL C00269 BC00269 V=8.3  +MOVJ EC00269
SMOVL C00270 BC00270 V=8.3  +MOVJ EC00270
SMOVL C00271 BC00271 V=8.3  +MOVJ EC00271
MOVL C00272 BC00272 V=8.3  +MOVJ EC00272 VJ=100.00
ARCOF
SMOVL C00273 BC00273 V=800.0  +MOVJ EC00273
SMOVL C00274 BC00274 V=1000.0  +MOVJ EC00274
SFTOF3D
'EndPath W4624
MOVJ C00275 BC00275 VJ=100.00  +MOVJ EC00275 VJ=100.00
'Path S4625
SFTOF3D
CALL JOB:CLEAN-R1_KM_NEW
MOVJ C00276 BC00276 VJ=100.00  +MOVJ EC00276 VJ=100.00
MOVJ C00277 BC00277 VJ=100.00  +MOVJ EC00277 VJ=100.00
MOVL C00278 BC00278 V=800.0  +MOVJ EC00278 VJ=100.00
SMOVL C00279 BC00279 V=166.7  +MOVJ EC00279
SREFP 3 C00280 BC00280  +REFP EC00280
CALL JOB:SEARCH-R1-S13D
SET P048 P006
SFTON3D P048
SMOVL C00281 BC00281 V=166.7  +MOVJ EC00281
SMOVL C00282 BC00282 V=166.7  +MOVJ EC00282
SREFP 3 C00283 BC00283  +REFP EC00283
CALL JOB:SEARCH-R1-S13D
SET P048 P006
SFTON3D P048
SMOVL C00284 BC00284 V=16.7  +MOVJ EC00284
MOVL C00285 BC00285 V=800.0  +MOVJ EC00285 VJ=100.00
MOVL C00286 BC00286 V=1000.0  +MOVJ EC00286 VJ=100.00
'EndPath S4625
'Path S4626
SFTOF3D
MOVJ C00287 BC00287 VJ=100.00  +MOVJ EC00287 VJ=100.00
MOVL C00288 BC00288 V=800.0  +MOVJ EC00288 VJ=100.00
SMOVL C00289 BC00289 V=166.7  +MOVJ EC00289
SREFP 3 C00290 BC00290  +REFP EC00290
CALL JOB:SEARCH-R1-S13D
SET P047 P006
SFTON3D P047
SMOVL C00291 BC00291 V=166.7  +MOVJ EC00291
SMOVL C00292 BC00292 V=166.7  +MOVJ EC00292
SREFP 3 C00293 BC00293  +REFP EC00293
CALL JOB:SEARCH-R1-S13D
SET P047 P006
SFTON3D P047
SMOVL C00294 BC00294 V=166.7  +MOVJ EC00294
MOVL C00295 BC00295 V=800.0  +MOVJ EC00295 VJ=100.00
MOVL C00296 BC00296 V=1000.0  +MOVJ EC00296 VJ=100.00
'EndPath S4626
MOVJ C00297 BC00297 VJ=100.00  +MOVJ EC00297 VJ=100.00
'Path S4627
SFTOF3D
MOVJ C00298 BC00298 VJ=100.00  +MOVJ EC00298 VJ=100.00
MOVL C00299 BC00299 V=800.0  +MOVJ EC00299 VJ=100.00
SMOVL C00300 BC00300 V=166.7  +MOVJ EC00300
SREFP 3 C00301 BC00301  +REFP EC00301
CALL JOB:SEARCH-R1-S13D
SET P046 P006
SFTON3D P046
SMOVL C00302 BC00302 V=166.7  +MOVJ EC00302
SREFP 3 C00303 BC00303  +REFP EC00303
CALL JOB:SEARCH-R1-S13D
SET P046 P006
SFTON3D P046
SMOVL C00304 BC00304 V=166.7  +MOVJ EC00304
MOVL C00305 BC00305 V=800.0  +MOVJ EC00305 VJ=100.00
'EndPath S4627
'Path S4628
SFTOF3D
MOVJ C00306 BC00306 VJ=100.00  +MOVJ EC00306 VJ=100.00
MOVJ C00307 BC00307 VJ=100.00  +MOVJ EC00307 VJ=100.00
MOVL C00308 BC00308 V=800.0  +MOVJ EC00308 VJ=100.00
SMOVL C00309 BC00309 V=166.7  +MOVJ EC00309
SREFP 3 C00310 BC00310  +REFP EC00310
CALL JOB:SEARCH-R1-S13D
SET P051 P006
SFTON3D P051
SMOVL C00311 BC00311 V=166.7  +MOVJ EC00311
SREFP 3 C00312 BC00312  +REFP EC00312
CALL JOB:SEARCH-R1-S13D
SET P051 P006
SFTON3D P051
SMOVL C00313 BC00313 V=166.7  +MOVJ EC00313
SMOVL C00314 BC00314 V=250.0  +MOVJ EC00314
SMOVL C00315 BC00315 V=166.7  +MOVJ EC00315
SREFP 3 C00316 BC00316  +REFP EC00316
CALL JOB:SEARCH-R1-S13D
SET P051 P006
SFTON3D P051
SMOVL C00317 BC00317 V=166.7  +MOVJ EC00317
MOVL C00318 BC00318 V=1000.0  +MOVJ EC00318 VJ=100.00
'EndPath S4629
'Path S4630
SFTOF3D
MOVJ C00319 BC00319 VJ=100.00  +MOVJ EC00319 VJ=100.00
MOVL C00320 BC00320 V=800.0  +MOVJ EC00320 VJ=100.00
SMOVL C00321 BC00321 V=166.7  +MOVJ EC00321
SREFP 3 C00322 BC00322  +REFP EC00322
CALL JOB:SEARCH-R1-S13D
SET P045 P006
SFTON3D P045
SMOVL C00323 BC00323 V=166.7  +MOVJ EC00323
SMOVL C00324 BC00324 V=166.7  +MOVJ EC00324
SREFP 3 C00325 BC00325  +REFP EC00325
CALL JOB:SEARCH-R1-S13D
SET P045 P006
SFTON3D P045
SMOVL C00326 BC00326 V=166.7  +MOVJ EC00326
MOVL C00327 BC00327 V=1000.0  +MOVJ EC00327 VJ=100.00
'EndPath S4630
'Path S4631
SFTOF3D
MOVJ C00328 BC00328 VJ=100.00  +MOVJ EC00328 VJ=100.00
MOVL C00329 BC00329 V=800.0  +MOVJ EC00329 VJ=100.00
SMOVL C00330 BC00330 V=166.7  +MOVJ EC00330
SREFP 3 C00331 BC00331  +REFP EC00331
CALL JOB:SEARCH-R1-S13D
SET P044 P006
SFTON3D P044
SMOVL C00332 BC00332 V=166.7  +MOVJ EC00332
SMOVL C00333 BC00333 V=166.7  +MOVJ EC00333
SREFP 3 C00334 BC00334  +REFP EC00334
CALL JOB:SEARCH-R1-S13D
SET P044 P006
SFTON3D P044
SMOVL C00335 BC00335 V=166.7  +MOVJ EC00335
MOVL C00336 BC00336 V=800.0  +MOVJ EC00336 VJ=100.00
MOVL C00337 BC00337 V=1000.0  +MOVJ EC00337 VJ=100.00
'EndPath S4631
'Path S4632
SFTOF3D
MOVJ C00338 BC00338 VJ=100.00  +MOVJ EC00338 VJ=100.00
MOVL C00339 BC00339 V=800.0  +MOVJ EC00339 VJ=100.00
SMOVL C00340 BC00340 V=166.7  +MOVJ EC00340
SREFP 3 C00341 BC00341  +REFP EC00341
CALL JOB:SEARCH-R1-S13D
SET P049 P006
SFTON3D P049
SMOVL C00342 BC00342 V=166.7  +MOVJ EC00342
SMOVL C00343 BC00343 V=800.0  +MOVJ EC00343
SMOVL C00344 BC00344 V=166.7  +MOVJ EC00344
SREFP 3 C00345 BC00345  +REFP EC00345
CALL JOB:SEARCH-R1-S13D
SET P049 P006
SFTON3D P049
SMOVL C00346 BC00346 V=166.7  +MOVJ EC00346
SFTOF3D
MOVL C00347 BC00347 V=1000.0  +MOVJ EC00347 VJ=100.00
'EndPath S4632
MOVJ C00348 BC00348 VJ=100.00  +MOVJ EC00348 VJ=100.00
MOVJ C00349 BC00349 VJ=50.00  +MOVJ EC00349 VJ=50.00
MOVJ C00350 BC00350 VJ=100.00  +MOVJ EC00350 VJ=100.00
MOVJ C00351 BC00351 VJ=100.00  +MOVJ EC00351 VJ=100.00
'Path S4633
SFTOF3D
MOVJ C00352 BC00352 VJ=100.00  +MOVJ EC00352 VJ=100.00
MOVL C00353 BC00353 V=800.0  +MOVJ EC00353 VJ=100.00
SMOVL C00354 BC00354 V=166.7  +MOVJ EC00354
SREFP 3 C00355 BC00355  +REFP EC00355
CALL JOB:SEARCH-R1-S13D
SET P043 P006
SFTON3D P043
SMOVL C00356 BC00356 V=166.7  +MOVJ EC00356
MOVL C00357 BC00357 V=800.0  +MOVJ EC00357 VJ=100.00
SMOVL C00358 BC00358 V=166.7  +MOVJ EC00358
SREFP 3 C00359 BC00359  +REFP EC00359
CALL JOB:SEARCH-R1-S13D
SET P043 P006
SFTON3D P043
SMOVL C00360 BC00360 V=166.7  +MOVJ EC00360
MOVL C00361 BC00361 V=1000.0  +MOVJ EC00361 VJ=100.00
'EndPath S4633
'Path S4634
SFTOF3D
MOVJ C00362 BC00362 VJ=100.00  +MOVJ EC00362 VJ=100.00
MOVL C00363 BC00363 V=800.0  +MOVJ EC00363 VJ=100.00
SMOVL C00364 BC00364 V=166.7  +MOVJ EC00364
SREFP 3 C00365 BC00365  +REFP EC00365
CALL JOB:SEARCH-R1-S13D
SET P042 P006
SFTON3D P042
SMOVL C00366 BC00366 V=166.7  +MOVJ EC00366
MOVL C00367 BC00367 V=800.0  +MOVJ EC00367 VJ=100.00
SMOVL C00368 BC00368 V=166.7  +MOVJ EC00368
SREFP 3 C00369 BC00369  +REFP EC00369
CALL JOB:SEARCH-R1-S13D
SET P042 P006
SFTON3D P042
SMOVL C00370 BC00370 V=166.7  +MOVJ EC00370
MOVL C00371 BC00371 V=1000.0  +MOVJ EC00371 VJ=100.00
'EndPath S4634
MOVJ C00372 BC00372 VJ=100.00  +MOVJ EC00372 VJ=100.00
MOVJ C00373 BC00373 VJ=100.00  +MOVJ EC00373 VJ=100.00
MOVJ C00374 BC00374 VJ=100.00  +MOVJ EC00374 VJ=100.00
MOVJ C00375 BC00375 VJ=100.00  +MOVJ EC00375 VJ=100.00
'Path W4635
SFTOF3D
SFTON3D P051
MOVJ C00376 BC00376 VJ=100.00  +MOVJ EC00376 VJ=100.00
SMOVL C00377 BC00377 V=800.0  +MOVJ EC00377
SMOVL C00378 BC00378 V=150.0 PL=0  +MOVJ EC00378
MACRO1 MJ#(0) ARGF14
SMOVL C00379 BC00379 V=11.7  +MOVJ EC00379
ARCOF
SMOVL C00380 BC00380 V=800.0  +MOVJ EC00380
SMOVL C00381 BC00381 V=1000.0  +MOVJ EC00381
MOVJ C00382 BC00382 VJ=100.00  +MOVJ EC00382 VJ=100.00
MOVJ C00383 BC00383 VJ=100.00  +MOVJ EC00383 VJ=100.00
SMOVL C00384 BC00384 V=250.0  +MOVJ EC00384
ARCON
SMOVL C00385 BC00385 V=11.7  +MOVJ EC00385
SMOVL C00386 BC00386 V=11.7  +MOVJ EC00386
ARCOF
SMOVL C00387 BC00387 V=166.7  +MOVJ EC00387
SMOVL C00388 BC00388 V=166.7  +MOVJ EC00388
SMOVL C00389 BC00389 V=166.7  +MOVJ EC00389
ARCON
SMOVL C00390 BC00390 V=9.2  +MOVJ EC00390
ARCOF
SMOVL C00391 BC00391 V=133.3  +MOVJ EC00391
SMOVL C00392 BC00392 V=666.7  +MOVJ EC00392
SFTOF3D
'EndPath W4635
'Path W4636
SFTOF3D
SFTON3D P045
MOVJ C00393 BC00393 VJ=100.00  +MOVJ EC00393 VJ=100.00
SMOVL C00394 BC00394 V=800.0  +MOVJ EC00394
SMOVL C00395 BC00395 V=150.0 PL=0  +MOVJ EC00395
MACRO1 MJ#(0) ARGF21
ARCON
SMOVL C00396 BC00396 V=11.7  +MOVJ EC00396
SMOVL C00397 BC00397 V=11.7  +MOVJ EC00397
ARCOF
SMOVL C00398 BC00398 V=800.0  +MOVJ EC00398
SMOVL C00399 BC00399 V=1000.0  +MOVJ EC00399
SFTOF3D
'EndPath W4636
'Path W4637
SFTOF3D
SFTON3D P045
MOVJ C00400 BC00400 VJ=100.00  +MOVJ EC00400 VJ=100.00
SMOVL C00401 BC00401 V=800.0  +MOVJ EC00401
SMOVL C00402 BC00402 V=150.0 PL=0  +MOVJ EC00402
ARCON
SMOVL C00403 BC00403 V=11.7  +MOVJ EC00403
SMOVL C00404 BC00404 V=11.7  +MOVJ EC00404
ARCOF
SMOVL C00405 BC00405 V=800.0  +MOVJ EC00405
SMOVL C00406 BC00406 V=1000.0  +MOVJ EC00406
SFTOF3D
'EndPath W4637
'Path W4638
SFTOF3D
SFTON3D P049
MOVJ C00407 BC00407 VJ=100.00  +MOVJ EC00407 VJ=100.00
SMOVL C00408 BC00408 V=800.0  +MOVJ EC00408
SMOVL C00409 BC00409 V=150.0 PL=0  +MOVJ EC00409
ARCON
SMOVL C00410 BC00410 V=10.0  +MOVJ EC00410
ARCOF
SMOVL C00411 BC00411 V=800.0  +MOVJ EC00411
SMOVL C00412 BC00412 V=1000.0  +MOVJ EC00412
SFTOF3D
'EndPath W4638
'Path W4639
SFTOF3D
MOVJ C00413 BC00413 VJ=20.00  +MOVJ EC00413 VJ=100.00
SMOVL C00414 BC00414 V=800.0  +MOVJ EC00414
SFTON3D P046
SMOVL C00415 BC00415 V=150.0 PL=0  +MOVJ EC00415
ARCON
SMOVL C00416 BC00416 V=11.7  +MOVJ EC00416
ARCOF
SMOVL C00417 BC00417 V=800.0  +MOVJ EC00417
SMOVL C00418 BC00418 V=1000.0  +MOVJ EC00418
SFTOF3D
'EndPath W4639
MOVJ C00419 BC00419 VJ=100.00  +MOVJ EC00419 VJ=100.00
'Path W4640
SFTOF3D
SFTON3D P048
MOVJ C00420 BC00420 VJ=100.00  +MOVJ EC00420 VJ=100.00
SMOVL C00421 BC00421 V=800.0  +MOVJ EC00421
SMOVL C00422 BC00422 V=150.0 PL=0  +MOVJ EC00422
ARCON
SMOVL C00423 BC00423 V=11.7  +MOVJ EC00423
ARCOF
SMOVL C00424 BC00424 V=800.0  +MOVJ EC00424
SMOVL C00425 BC00425 V=1000.0  +MOVJ EC00425
SFTOF3D
'EndPath W4640
'Path W4641
SFTOF3D
SFTON3D P048
SMOVL C00426 BC00426 V=150.0 PL=0  +MOVJ EC00426
ARCON
SMOVL C00427 BC00427 V=11.7  +MOVJ EC00427
ARCOF
SFTOF3D
SMOVL C00428 BC00428 V=800.0  +MOVJ EC00428
SFTOF3D
'EndPath W4641
'Path W4642
SFTOF3D
SFTON3D P047
MOVJ C00429 BC00429 VJ=100.00  +MOVJ EC00429 VJ=100.00
SMOVL C00430 BC00430 V=800.0  +MOVJ EC00430
SMOVL C00431 BC00431 V=150.0 PL=0  +MOVJ EC00431
ARCON
SMOVL C00432 BC00432 V=11.7  +MOVJ EC00432
ARCOF
SMOVL C00433 BC00433 V=800.0  +MOVJ EC00433
SMOVL C00434 BC00434 V=1000.0  +MOVJ EC00434
SFTOF3D
'EndPath W4642
MOVJ C00435 BC00435 VJ=100.00  +MOVJ EC00435 VJ=100.00
MOVJ C00436 BC00436 VJ=100.00  +MOVJ EC00436 VJ=100.00
'Path W4643
SFTOF3D
SFTON3D P043
MOVJ C00437 BC00437 VJ=100.00  +MOVJ EC00437 VJ=100.00
SMOVL C00438 BC00438 V=800.0  +MOVJ EC00438
SMOVL C00439 BC00439 V=150.0 PL=0  +MOVJ EC00439
ARCON
SMOVL C00440 BC00440 V=11.7  +MOVJ EC00440
ARCOF
SMOVL C00441 BC00441 V=800.0  +MOVJ EC00441
SMOVL C00442 BC00442 V=1000.0  +MOVJ EC00442
SFTOF3D
'EndPath W4643
'Path W4644
SFTOF3D
SFTON3D P043
SMOVL C00443 BC00443 V=150.0 PL=0  +MOVJ EC00443
ARCON
SMOVL C00444 BC00444 V=11.7  +MOVJ EC00444
ARCOF
SMOVL C00445 BC00445 V=800.0  +MOVJ EC00445
SFTOF3D
'EndPath W4644
'Path W4645
SFTOF3D
SFTON3D P042
MOVJ C00446 BC00446 VJ=100.00  +MOVJ EC00446 VJ=100.00
SMOVL C00447 BC00447 V=800.0  +MOVJ EC00447
SMOVL C00448 BC00448 V=150.0 PL=0  +MOVJ EC00448
ARCON
SMOVL C00449 BC00449 V=11.7  +MOVJ EC00449
ARCOF
SMOVL C00450 BC00450 V=800.0  +MOVJ EC00450
SMOVL C00451 BC00451 V=1000.0  +MOVJ EC00451
SFTOF3D
'EndPath W4645
'Path W4646
SFTOF3D
SFTON3D P042
MOVJ C00452 BC00452 VJ=100.00  +MOVJ EC00452 VJ=100.00
SMOVL C00453 BC00453 V=800.0  +MOVJ EC00453
SMOVL C00454 BC00454 V=150.0 PL=0  +MOVJ EC00454
ARCON
SMOVL C00455 BC00455 V=11.7  +MOVJ EC00455
ARCOF
SMOVL C00456 BC00456 V=800.0  +MOVJ EC00456
SMOVL C00457 BC00457 V=1000.0  +MOVJ EC00457
SFTOF3D
'EndPath W4646
'3
MOVJ C00458 BC00458 VJ=100.00  +MOVJ EC00458 VJ=100.00
MOVJ C00459 BC00459 VJ=100.00  +MOVJ EC00459 VJ=100.00
MOVJ C00460 BC00460 VJ=20.00  +MOVJ EC00460 VJ=20.00
'Path W4647
SFTOF3D
SFTON3D P044
MOVJ C00461 BC00461 VJ=100.00  +MOVJ EC00461 VJ=100.00
SMOVL C00462 BC00462 V=800.0  +MOVJ EC00462
SMOVL C00463 BC00463 V=150.0 PL=0  +MOVJ EC00463
ARCON
SMOVL C00464 BC00464 V=11.7  +MOVJ EC00464
ARCOF
SMOVL C00465 BC00465 V=800.0  +MOVJ EC00465
SMOVL C00466 BC00466 V=1000.0  +MOVJ EC00466
SFTOF3D
'EndPath W4647
'Path W4648
SFTOF3D
SFTON3D P046
MOVJ C00467 BC00467 VJ=100.00  +MOVJ EC00467 VJ=100.00
SMOVL C00468 BC00468 V=800.0  +MOVJ EC00468
SMOVL C00469 BC00469 V=150.0 PL=0  +MOVJ EC00469
MACRO1 MJ#(0) ARGF14
ARCON
SMOVL C00470 BC00470 V=11.7  +MOVJ EC00470
ARCOF
SMOVL C00471 BC00471 V=800.0  +MOVJ EC00471
SMOVL C00472 BC00472 V=1000.0  +MOVJ EC00472
SFTOF3D
'EndPath W4648
MOVJ C00473 BC00473 VJ=100.00  +MOVJ EC00473 VJ=100.00
MOVJ C00474 BC00474 VJ=100.00  +MOVJ EC00474 VJ=100.00
END
